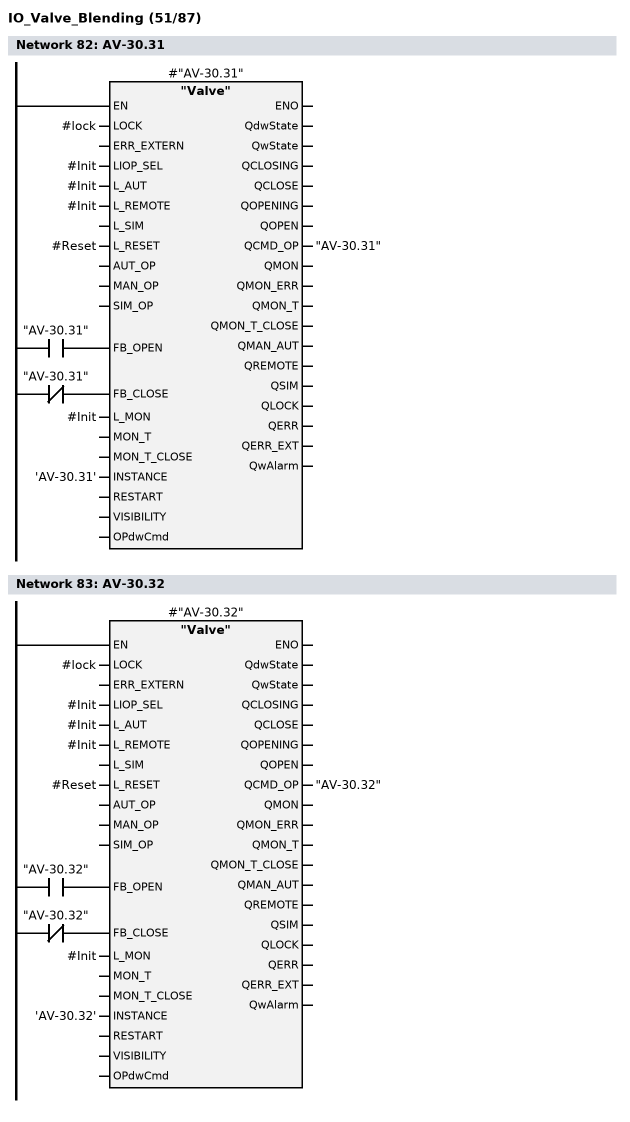
   RUNG wire#powerrail
      #"AV-30.31"(FB_OPEN := wire#w1, FB_CLOSE := wire#w2, LOCK := #lock, ERR_EXTERN :=, LIOP_SEL := #Init, L_AUT := #Init, L_REMOTE := #Init, L_SIM :=, L_RESET := #Reset, AUT_OP :=, MAN_OP :=, SIM_OP :=, L_MON := #Init, MON_T :=, MON_T_CLOSE :=, INSTANCE := 'AV-30.31', RESTART :=, VISIBILITY :=, OPdwCmd :=, QdwState =>, QwState =>, QCLOSING =>, QCLOSE =>, QOPENING =>, QOPEN =>, QCMD_OP => "AV-30.31", QMON =>, QMON_ERR =>, QMON_T =>, QMON_T_CLOSE =>, QMAN_AUT =>, QREMOTE =>, QSIM =>, QLOCK =>, QERR =>, QERR_EXT =>, QwAlarm =>)
   END_RUNG
   RUNG wire#powerrail
      Contact( "AV-30.31" )
   END_RUNG wire#w1
   RUNG wire#powerrail
      I_Contact( "AV-30.31" )
   END_RUNG wire#w2
   // the same network as SCL:
   #"AV-30.31"(LOCK := #lock,   // "Valve"
               LIOP_SEL := #Init,
               L_AUT := #Init,
               L_REMOTE := #Init,
               L_RESET := #Reset,
               FB_OPEN := "AV-30.31",
               FB_CLOSE := NOT "AV-30.31",
               L_MON := #Init,
               INSTANCE := 'AV-30.31',
               QCMD_OP => "AV-30.31");
END_REGION

REGION Network 83: AV-30.32
   RUNG wire#powerrail
      #"AV-30.32"(FB_OPEN := wire#w1, FB_CLOSE := wire#w2, LOCK := #lock, ERR_EXTERN :=, LIOP_SEL := #Init, L_AUT := #Init, L_REMOTE := #Init, L_SIM :=, L_RESET := #Reset, AUT_OP :=, MAN_OP :=, SIM_OP :=, L_MON := #Init, MON_T :=, MON_T_CLOSE :=, INSTANCE := 'AV-30.32', RESTART :=, VISIBILITY :=, OPdwCmd :=, QdwState =>, QwState =>, QCLOSING =>, QCLOSE =>, QOPENING =>, QOPEN =>, QCMD_OP => "AV-30.32", QMON =>, QMON_ERR =>, QMON_T =>, QMON_T_CLOSE =>, QMAN_AUT =>, QREMOTE =>, QSIM =>, QLOCK =>, QERR =>, QERR_EXT =>, QwAlarm =>)
   END_RUNG
   RUNG wire#powerrail
      Contact( "AV-30.32" )
   END_RUNG wire#w1
   RUNG wire#powerrail
      I_Contact( "AV-30.32" )
   END_RUNG wire#w2
   // the same network as SCL:
   #"AV-30.32"(LOCK := #lock,   // "Valve"
               LIOP_SEL := #Init,
               L_AUT := #Init,
               L_REMOTE := #Init,
               L_RESET := #Reset,
               FB_OPEN := "AV-30.32",
               FB_CLOSE := NOT "AV-30.32",
               L_MON := #Init,
               INSTANCE := 'AV-30.32',
               QCMD_OP => "AV-30.32");
END_REGION

REGION Network 84: AV-30.33
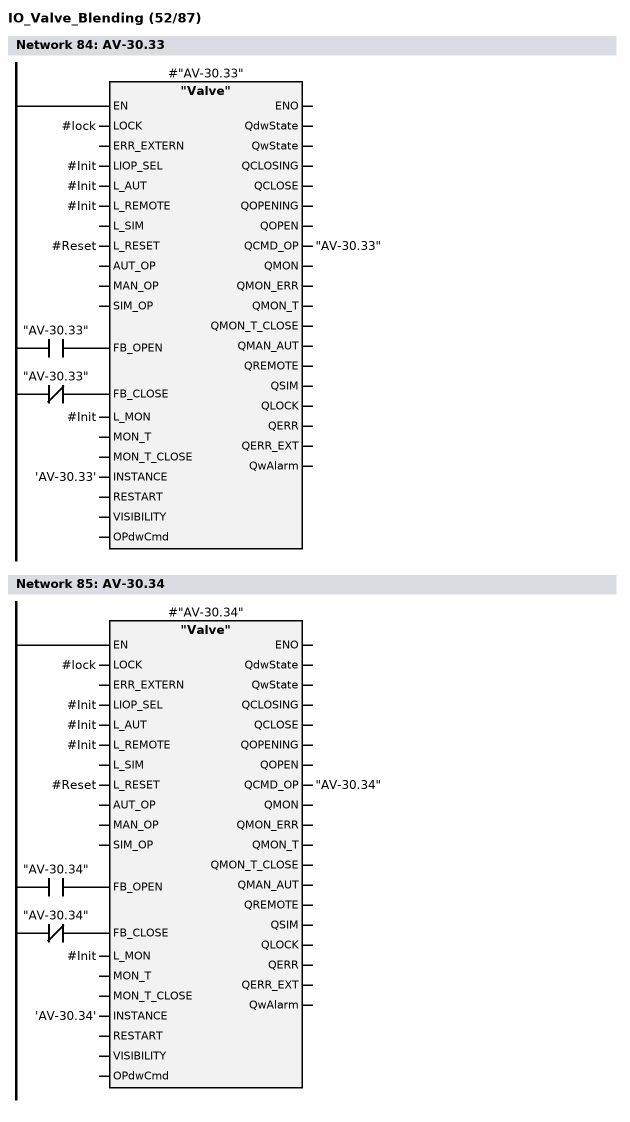
   RUNG wire#powerrail
      #"AV-30.33"(FB_OPEN := wire#w1, FB_CLOSE := wire#w2, LOCK := #lock, ERR_EXTERN :=, LIOP_SEL := #Init, L_AUT := #Init, L_REMOTE := #Init, L_SIM :=, L_RESET := #Reset, AUT_OP :=, MAN_OP :=, SIM_OP :=, L_MON := #Init, MON_T :=, MON_T_CLOSE :=, INSTANCE := 'AV-30.33', RESTART :=, VISIBILITY :=, OPdwCmd :=, QdwState =>, QwState =>, QCLOSING =>, QCLOSE =>, QOPENING =>, QOPEN =>, QCMD_OP => "AV-30.33", QMON =>, QMON_ERR =>, QMON_T =>, QMON_T_CLOSE =>, QMAN_AUT =>, QREMOTE =>, QSIM =>, QLOCK =>, QERR =>, QERR_EXT =>, QwAlarm =>)
   END_RUNG
   RUNG wire#powerrail
      Contact( "AV-30.33" )
   END_RUNG wire#w1
   RUNG wire#powerrail
      I_Contact( "AV-30.33" )
   END_RUNG wire#w2
   // the same network as SCL:
   #"AV-30.33"(LOCK := #lock,   // "Valve"
               LIOP_SEL := #Init,
               L_AUT := #Init,
               L_REMOTE := #Init,
               L_RESET := #Reset,
               FB_OPEN := "AV-30.33",
               FB_CLOSE := NOT "AV-30.33",
               L_MON := #Init,
               INSTANCE := 'AV-30.33',
               QCMD_OP => "AV-30.33");
END_REGION

REGION Network 85: AV-30.34
   RUNG wire#powerrail
      #"AV-30.34"(FB_OPEN := wire#w1, FB_CLOSE := wire#w2, LOCK := #lock, ERR_EXTERN :=, LIOP_SEL := #Init, L_AUT := #Init, L_REMOTE := #Init, L_SIM :=, L_RESET := #Reset, AUT_OP :=, MAN_OP :=, SIM_OP :=, L_MON := #Init, MON_T :=, MON_T_CLOSE :=, INSTANCE := 'AV-30.34', RESTART :=, VISIBILITY :=, OPdwCmd :=, QdwState =>, QwState =>, QCLOSING =>, QCLOSE =>, QOPENING =>, QOPEN =>, QCMD_OP => "AV-30.34", QMON =>, QMON_ERR =>, QMON_T =>, QMON_T_CLOSE =>, QMAN_AUT =>, QREMOTE =>, QSIM =>, QLOCK =>, QERR =>, QERR_EXT =>, QwAlarm =>)
   END_RUNG
   RUNG wire#powerrail
      Contact( "AV-30.34" )
   END_RUNG wire#w1
   RUNG wire#powerrail
      I_Contact( "AV-30.34" )
   END_RUNG wire#w2
   // the same network as SCL:
   #"AV-30.34"(LOCK := #lock,   // "Valve"
               LIOP_SEL := #Init,
               L_AUT := #Init,
               L_REMOTE := #Init,
               L_RESET := #Reset,
               FB_OPEN := "AV-30.34",
               FB_CLOSE := NOT "AV-30.34",
               L_MON := #Init,
               INSTANCE := 'AV-30.34',
               QCMD_OP => "AV-30.34");
END_REGION

REGION Network 86: AV-30.35
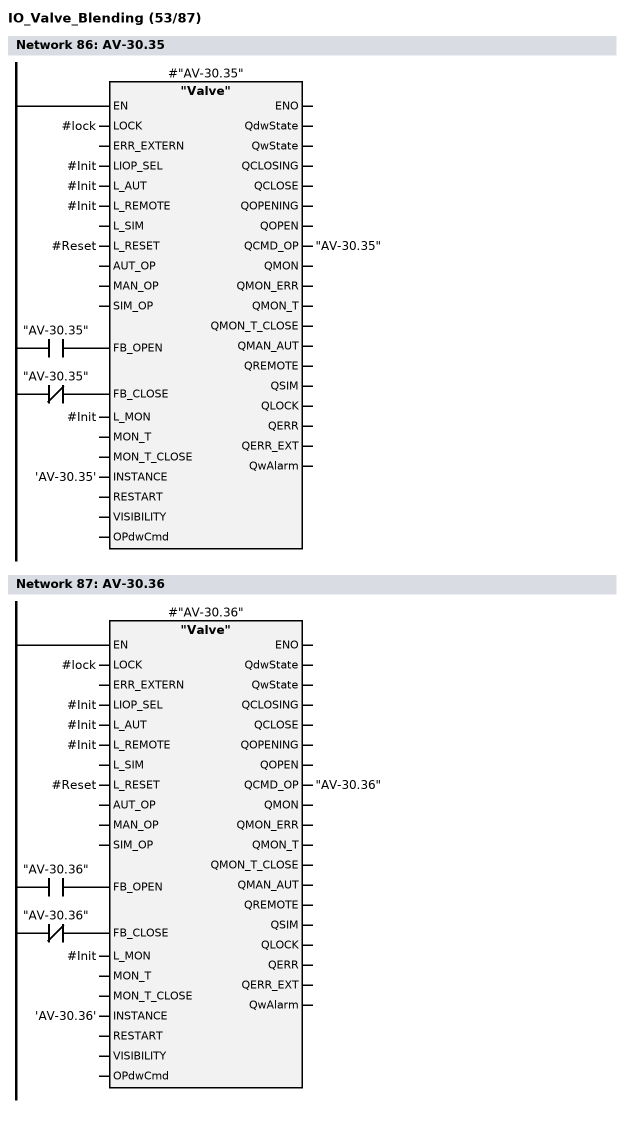
   RUNG wire#powerrail
      #"AV-30.35"(FB_OPEN := wire#w1, FB_CLOSE := wire#w2, LOCK := #lock, ERR_EXTERN :=, LIOP_SEL := #Init, L_AUT := #Init, L_REMOTE := #Init, L_SIM :=, L_RESET := #Reset, AUT_OP :=, MAN_OP :=, SIM_OP :=, L_MON := #Init, MON_T :=, MON_T_CLOSE :=, INSTANCE := 'AV-30.35', RESTART :=, VISIBILITY :=, OPdwCmd :=, QdwState =>, QwState =>, QCLOSING =>, QCLOSE =>, QOPENING =>, QOPEN =>, QCMD_OP => "AV-30.35", QMON =>, QMON_ERR =>, QMON_T =>, QMON_T_CLOSE =>, QMAN_AUT =>, QREMOTE =>, QSIM =>, QLOCK =>, QERR =>, QERR_EXT =>, QwAlarm =>)
   END_RUNG
   RUNG wire#powerrail
      Contact( "AV-30.35" )
   END_RUNG wire#w1
   RUNG wire#powerrail
      I_Contact( "AV-30.35" )
   END_RUNG wire#w2
   // the same network as SCL:
   #"AV-30.35"(LOCK := #lock,   // "Valve"
               LIOP_SEL := #Init,
               L_AUT := #Init,
               L_REMOTE := #Init,
               L_RESET := #Reset,
               FB_OPEN := "AV-30.35",
               FB_CLOSE := NOT "AV-30.35",
               L_MON := #Init,
               INSTANCE := 'AV-30.35',
               QCMD_OP => "AV-30.35");
END_REGION

REGION Network 87: AV-30.36
   RUNG wire#powerrail
      #"AV-30.36"(FB_OPEN := wire#w1, FB_CLOSE := wire#w2, LOCK := #lock, ERR_EXTERN :=, LIOP_SEL := #Init, L_AUT := #Init, L_REMOTE := #Init, L_SIM :=, L_RESET := #Reset, AUT_OP :=, MAN_OP :=, SIM_OP :=, L_MON := #Init, MON_T :=, MON_T_CLOSE :=, INSTANCE := 'AV-30.36', RESTART :=, VISIBILITY :=, OPdwCmd :=, QdwState =>, QwState =>, QCLOSING =>, QCLOSE =>, QOPENING =>, QOPEN =>, QCMD_OP => "AV-30.36", QMON =>, QMON_ERR =>, QMON_T =>, QMON_T_CLOSE =>, QMAN_AUT =>, QREMOTE =>, QSIM =>, QLOCK =>, QERR =>, QERR_EXT =>, QwAlarm =>)
   END_RUNG
   RUNG wire#powerrail
      Contact( "AV-30.36" )
   END_RUNG wire#w1
   RUNG wire#powerrail
      I_Contact( "AV-30.36" )
   END_RUNG wire#w2
   // the same network as SCL:
   #"AV-30.36"(LOCK := #lock,   // "Valve"
               LIOP_SEL := #Init,
               L_AUT := #Init,
               L_REMOTE := #Init,
               L_RESET := #Reset,
               FB_OPEN := "AV-30.36",
               FB_CLOSE := NOT "AV-30.36",
               L_MON := #Init,
               INSTANCE := 'AV-30.36',
               QCMD_OP => "AV-30.36");
END_REGION

REGION Network 88: AV-30.37
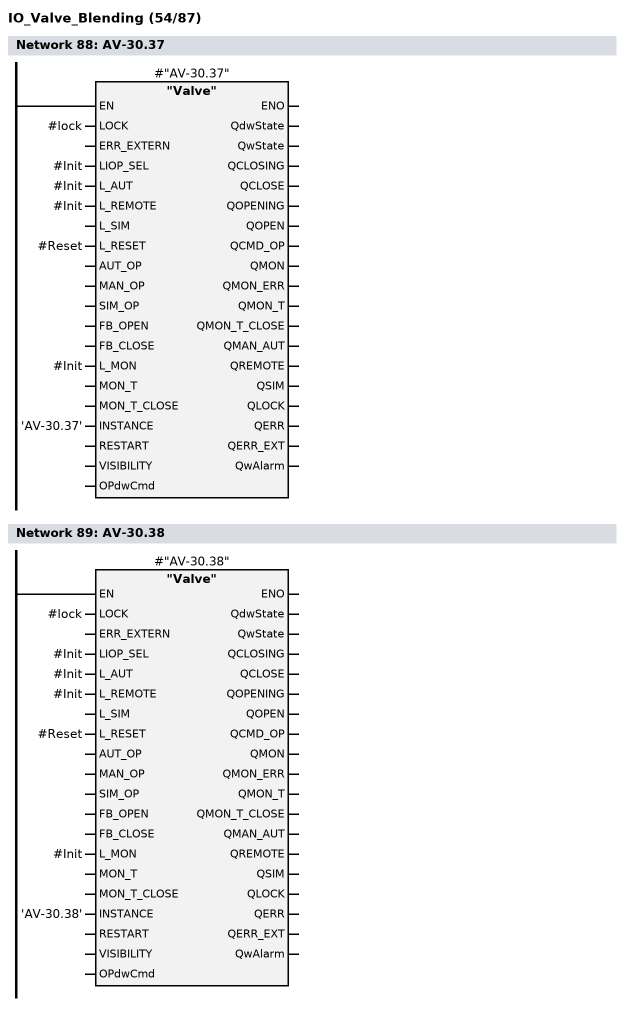
   RUNG wire#powerrail
      #"AV-30.37"(LOCK := #lock, ERR_EXTERN :=, LIOP_SEL := #Init, L_AUT := #Init, L_REMOTE := #Init, L_SIM :=, L_RESET := #Reset, AUT_OP :=, MAN_OP :=, SIM_OP :=, FB_OPEN :=, FB_CLOSE :=, L_MON := #Init, MON_T :=, MON_T_CLOSE :=, INSTANCE := 'AV-30.37', RESTART :=, VISIBILITY :=, OPdwCmd :=, QdwState =>, QwState =>, QCLOSING =>, QCLOSE =>, QOPENING =>, QOPEN =>, QCMD_OP =>, QMON =>, QMON_ERR =>, QMON_T =>, QMON_T_CLOSE =>, QMAN_AUT =>, QREMOTE =>, QSIM =>, QLOCK =>, QERR =>, QERR_EXT =>, QwAlarm =>)
   END_RUNG
   // the same network as SCL:
   #"AV-30.37"(LOCK := #lock,   // "Valve"
               LIOP_SEL := #Init,
               L_AUT := #Init,
               L_REMOTE := #Init,
               L_RESET := #Reset,
               L_MON := #Init,
               INSTANCE := 'AV-30.37');
END_REGION

REGION Network 89: AV-30.38
   RUNG wire#powerrail
      #"AV-30.38"(LOCK := #lock, ERR_EXTERN :=, LIOP_SEL := #Init, L_AUT := #Init, L_REMOTE := #Init, L_SIM :=, L_RESET := #Reset, AUT_OP :=, MAN_OP :=, SIM_OP :=, FB_OPEN :=, FB_CLOSE :=, L_MON := #Init, MON_T :=, MON_T_CLOSE :=, INSTANCE := 'AV-30.38', RESTART :=, VISIBILITY :=, OPdwCmd :=, QdwState =>, QwState =>, QCLOSING =>, QCLOSE =>, QOPENING =>, QOPEN =>, QCMD_OP =>, QMON =>, QMON_ERR =>, QMON_T =>, QMON_T_CLOSE =>, QMAN_AUT =>, QREMOTE =>, QSIM =>, QLOCK =>, QERR =>, QERR_EXT =>, QwAlarm =>)
   END_RUNG
   // the same network as SCL:
   #"AV-30.38"(LOCK := #lock,   // "Valve"
               LIOP_SEL := #Init,
               L_AUT := #Init,
               L_REMOTE := #Init,
               L_RESET := #Reset,
               L_MON := #Init,
               INSTANCE := 'AV-30.38');
END_REGION

REGION Network 90: AV-30.39
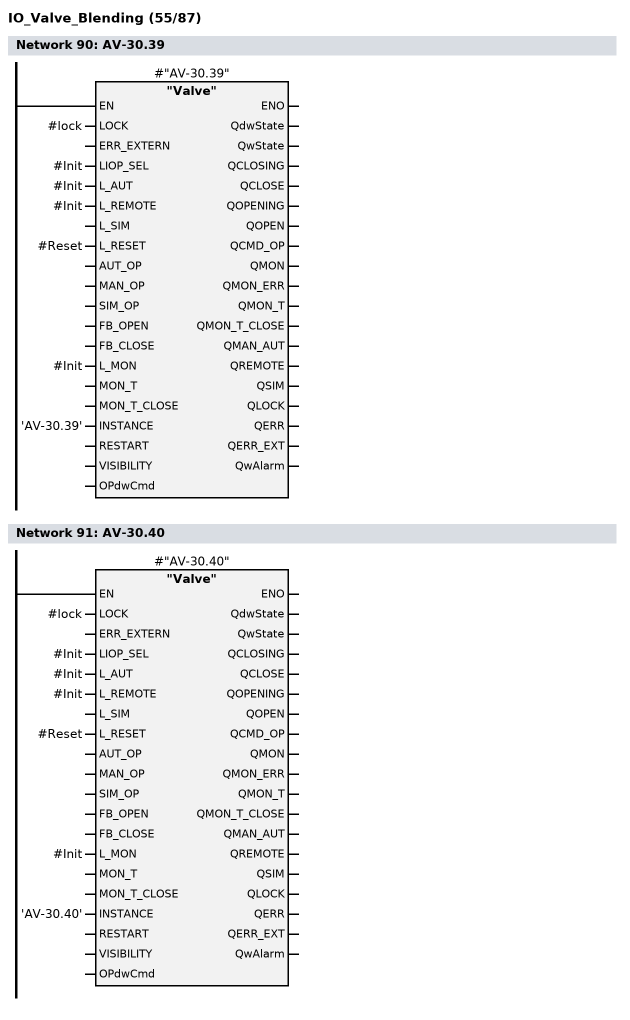
   RUNG wire#powerrail
      #"AV-30.39"(LOCK := #lock, ERR_EXTERN :=, LIOP_SEL := #Init, L_AUT := #Init, L_REMOTE := #Init, L_SIM :=, L_RESET := #Reset, AUT_OP :=, MAN_OP :=, SIM_OP :=, FB_OPEN :=, FB_CLOSE :=, L_MON := #Init, MON_T :=, MON_T_CLOSE :=, INSTANCE := 'AV-30.39', RESTART :=, VISIBILITY :=, OPdwCmd :=, QdwState =>, QwState =>, QCLOSING =>, QCLOSE =>, QOPENING =>, QOPEN =>, QCMD_OP =>, QMON =>, QMON_ERR =>, QMON_T =>, QMON_T_CLOSE =>, QMAN_AUT =>, QREMOTE =>, QSIM =>, QLOCK =>, QERR =>, QERR_EXT =>, QwAlarm =>)
   END_RUNG
   // the same network as SCL:
   #"AV-30.39"(LOCK := #lock,   // "Valve"
               LIOP_SEL := #Init,
               L_AUT := #Init,
               L_REMOTE := #Init,
               L_RESET := #Reset,
               L_MON := #Init,
               INSTANCE := 'AV-30.39');
END_REGION

REGION Network 91: AV-30.40
   RUNG wire#powerrail
      #"AV-30.40"(LOCK := #lock, ERR_EXTERN :=, LIOP_SEL := #Init, L_AUT := #Init, L_REMOTE := #Init, L_SIM :=, L_RESET := #Reset, AUT_OP :=, MAN_OP :=, SIM_OP :=, FB_OPEN :=, FB_CLOSE :=, L_MON := #Init, MON_T :=, MON_T_CLOSE :=, INSTANCE := 'AV-30.40', RESTART :=, VISIBILITY :=, OPdwCmd :=, QdwState =>, QwState =>, QCLOSING =>, QCLOSE =>, QOPENING =>, QOPEN =>, QCMD_OP =>, QMON =>, QMON_ERR =>, QMON_T =>, QMON_T_CLOSE =>, QMAN_AUT =>, QREMOTE =>, QSIM =>, QLOCK =>, QERR =>, QERR_EXT =>, QwAlarm =>)
   END_RUNG
   // the same network as SCL:
   #"AV-30.40"(LOCK := #lock,   // "Valve"
               LIOP_SEL := #Init,
               L_AUT := #Init,
               L_REMOTE := #Init,
               L_RESET := #Reset,
               L_MON := #Init,
               INSTANCE := 'AV-30.40');
END_REGION

REGION Network 92: AV-30.41
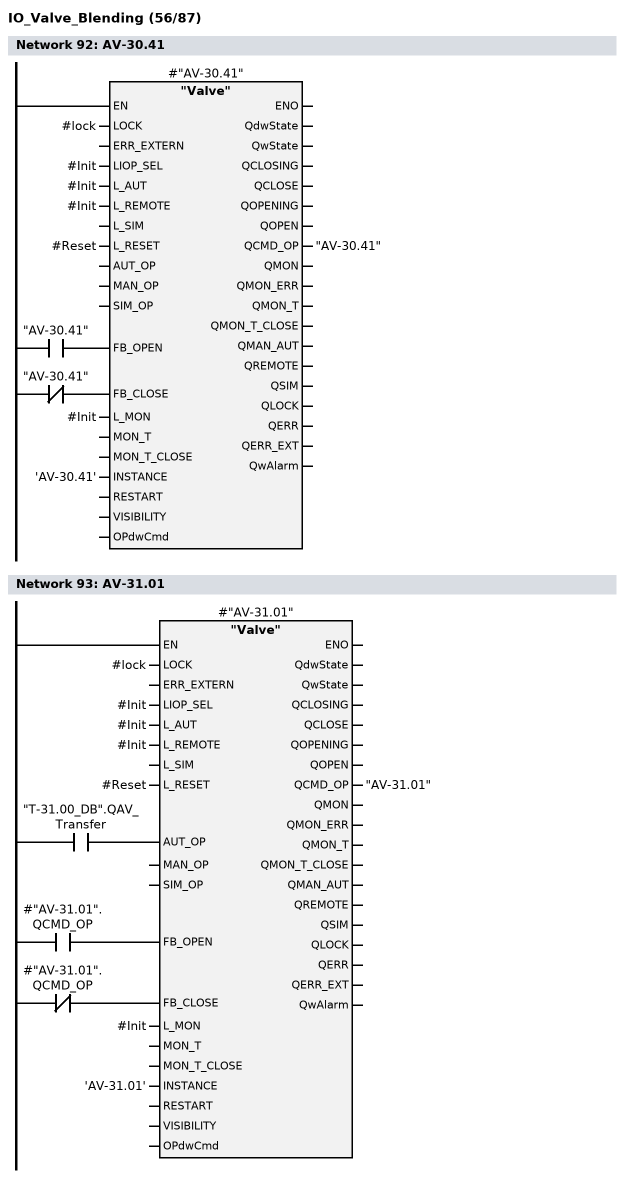
   RUNG wire#powerrail
      #"AV-30.41"(FB_OPEN := wire#w1, FB_CLOSE := wire#w2, LOCK := #lock, ERR_EXTERN :=, LIOP_SEL := #Init, L_AUT := #Init, L_REMOTE := #Init, L_SIM :=, L_RESET := #Reset, AUT_OP :=, MAN_OP :=, SIM_OP :=, L_MON := #Init, MON_T :=, MON_T_CLOSE :=, INSTANCE := 'AV-30.41', RESTART :=, VISIBILITY :=, OPdwCmd :=, QdwState =>, QwState =>, QCLOSING =>, QCLOSE =>, QOPENING =>, QOPEN =>, QCMD_OP => "AV-30.41", QMON =>, QMON_ERR =>, QMON_T =>, QMON_T_CLOSE =>, QMAN_AUT =>, QREMOTE =>, QSIM =>, QLOCK =>, QERR =>, QERR_EXT =>, QwAlarm =>)
   END_RUNG
   RUNG wire#powerrail
      Contact( "AV-30.41" )
   END_RUNG wire#w1
   RUNG wire#powerrail
      I_Contact( "AV-30.41" )
   END_RUNG wire#w2
   // the same network as SCL:
   #"AV-30.41"(LOCK := #lock,   // "Valve"
               LIOP_SEL := #Init,
               L_AUT := #Init,
               L_REMOTE := #Init,
               L_RESET := #Reset,
               FB_OPEN := "AV-30.41",
               FB_CLOSE := NOT "AV-30.41",
               L_MON := #Init,
               INSTANCE := 'AV-30.41',
               QCMD_OP => "AV-30.41");
END_REGION

REGION Network 93: AV-31.01
   RUNG wire#powerrail
      #"AV-31.01"(AUT_OP := wire#w1, FB_OPEN := wire#w2, FB_CLOSE := wire#w3, LOCK := #lock, ERR_EXTERN :=, LIOP_SEL := #Init, L_AUT := #Init, L_REMOTE := #Init, L_SIM :=, L_RESET := #Reset, MAN_OP :=, SIM_OP :=, L_MON := #Init, MON_T :=, MON_T_CLOSE :=, INSTANCE := 'AV-31.01', RESTART :=, VISIBILITY :=, OPdwCmd :=, QdwState =>, QwState =>, QCLOSING =>, QCLOSE =>, QOPENING =>, QOPEN =>, QCMD_OP => "AV-31.01", QMON =>, QMON_ERR =>, QMON_T =>, QMON_T_CLOSE =>, QMAN_AUT =>, QREMOTE =>, QSIM =>, QLOCK =>, QERR =>, QERR_EXT =>, QwAlarm =>)
   END_RUNG
   RUNG wire#powerrail
      Contact( "T-31.00_DB".QAV_Transfer )
   END_RUNG wire#w1
   RUNG wire#powerrail
      Contact( #"AV-31.01".QCMD_OP )
   END_RUNG wire#w2
   RUNG wire#powerrail
      I_Contact( #"AV-31.01".QCMD_OP )
   END_RUNG wire#w3
   // the same network as SCL:
   #"AV-31.01"(LOCK := #lock,   // "Valve"
               LIOP_SEL := #Init,
               L_AUT := #Init,
               L_REMOTE := #Init,
               L_RESET := #Reset,
               AUT_OP := "T-31.00_DB".QAV_Transfer,
               FB_OPEN := #"AV-31.01".QCMD_OP,
               FB_CLOSE := NOT #"AV-31.01".QCMD_OP,
               L_MON := #Init,
               INSTANCE := 'AV-31.01',
               QCMD_OP => "AV-31.01");
END_REGION

REGION Network 94: AV-31.02
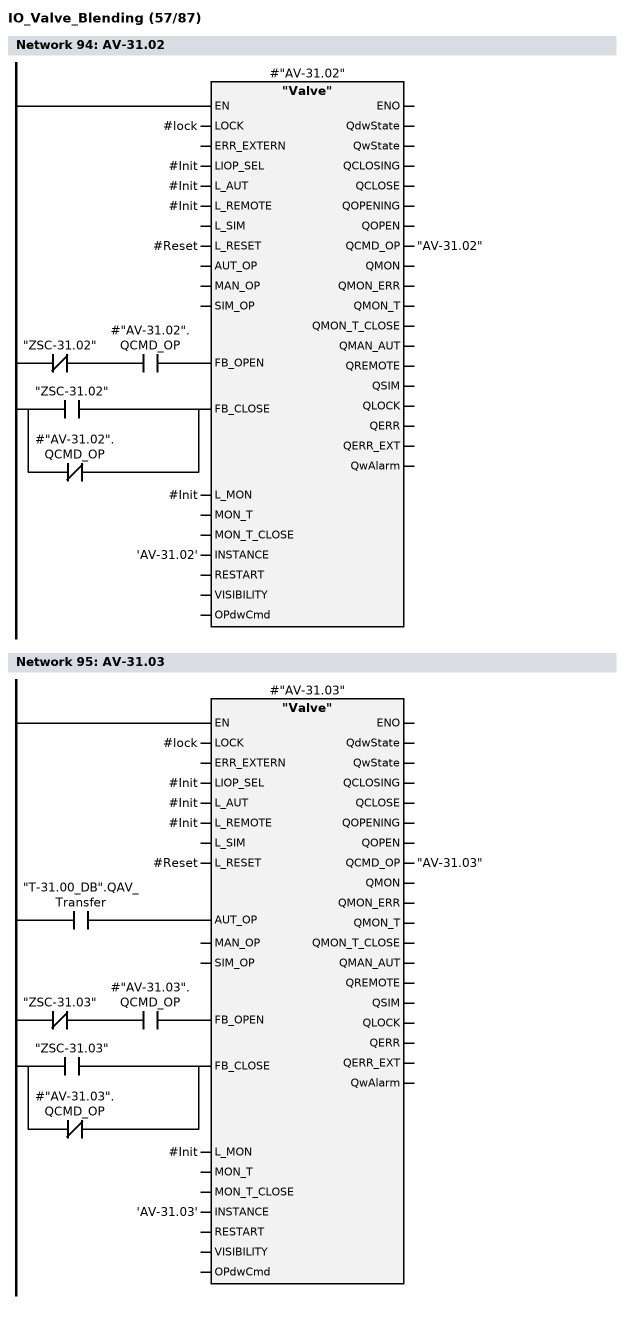
   RUNG wire#powerrail
      #"AV-31.02"(FB_OPEN := wire#w1, FB_CLOSE := wire#w2, LOCK := #lock, ERR_EXTERN :=, LIOP_SEL := #Init, L_AUT := #Init, L_REMOTE := #Init, L_SIM :=, L_RESET := #Reset, AUT_OP :=, MAN_OP :=, SIM_OP :=, L_MON := #Init, MON_T :=, MON_T_CLOSE :=, INSTANCE := 'AV-31.02', RESTART :=, VISIBILITY :=, OPdwCmd :=, QdwState =>, QwState =>, QCLOSING =>, QCLOSE =>, QOPENING =>, QOPEN =>, QCMD_OP => "AV-31.02", QMON =>, QMON_ERR =>, QMON_T =>, QMON_T_CLOSE =>, QMAN_AUT =>, QREMOTE =>, QSIM =>, QLOCK =>, QERR =>, QERR_EXT =>, QwAlarm =>)
   END_RUNG
   RUNG wire#powerrail
      I_Contact( "ZSC-31.02" )
      Contact( #"AV-31.02".QCMD_OP )
   END_RUNG wire#w1
   RUNG wire#powerrail
      Contact( "ZSC-31.02" )
   END_RUNG wire#w2
   RUNG wire#powerrail
      I_Contact( #"AV-31.02".QCMD_OP )
   END_RUNG wire#w2
   // the same network as SCL:
   #"AV-31.02"(LOCK := #lock,   // "Valve"
               LIOP_SEL := #Init,
               L_AUT := #Init,
               L_REMOTE := #Init,
               L_RESET := #Reset,
               FB_OPEN := NOT "ZSC-31.02" AND #"AV-31.02".QCMD_OP,
               FB_CLOSE := "ZSC-31.02" OR NOT #"AV-31.02".QCMD_OP,
               L_MON := #Init,
               INSTANCE := 'AV-31.02',
               QCMD_OP => "AV-31.02");
END_REGION

REGION Network 95: AV-31.03
   RUNG wire#powerrail
      #"AV-31.03"(AUT_OP := wire#w1, FB_OPEN := wire#w2, FB_CLOSE := wire#w3, LOCK := #lock, ERR_EXTERN :=, LIOP_SEL := #Init, L_AUT := #Init, L_REMOTE := #Init, L_SIM :=, L_RESET := #Reset, MAN_OP :=, SIM_OP :=, L_MON := #Init, MON_T :=, MON_T_CLOSE :=, INSTANCE := 'AV-31.03', RESTART :=, VISIBILITY :=, OPdwCmd :=, QdwState =>, QwState =>, QCLOSING =>, QCLOSE =>, QOPENING =>, QOPEN =>, QCMD_OP => "AV-31.03", QMON =>, QMON_ERR =>, QMON_T =>, QMON_T_CLOSE =>, QMAN_AUT =>, QREMOTE =>, QSIM =>, QLOCK =>, QERR =>, QERR_EXT =>, QwAlarm =>)
   END_RUNG
   RUNG wire#powerrail
      Contact( "T-31.00_DB".QAV_Transfer )
   END_RUNG wire#w1
   RUNG wire#powerrail
      I_Contact( "ZSC-31.03" )
      Contact( #"AV-31.03".QCMD_OP )
   END_RUNG wire#w2
   RUNG wire#powerrail
      Contact( "ZSC-31.03" )
   END_RUNG wire#w3
   RUNG wire#powerrail
      I_Contact( #"AV-31.03".QCMD_OP )
   END_RUNG wire#w3
   // the same network as SCL:
   #"AV-31.03"(LOCK := #lock,   // "Valve"
               LIOP_SEL := #Init,
               L_AUT := #Init,
               L_REMOTE := #Init,
               L_RESET := #Reset,
               AUT_OP := "T-31.00_DB".QAV_Transfer,
               FB_OPEN := NOT "ZSC-31.03" AND #"AV-31.03".QCMD_OP,
               FB_CLOSE := "ZSC-31.03" OR NOT #"AV-31.03".QCMD_OP,
               L_MON := #Init,
               INSTANCE := 'AV-31.03',
               QCMD_OP => "AV-31.03");
END_REGION

REGION Network 96: AV-31.04
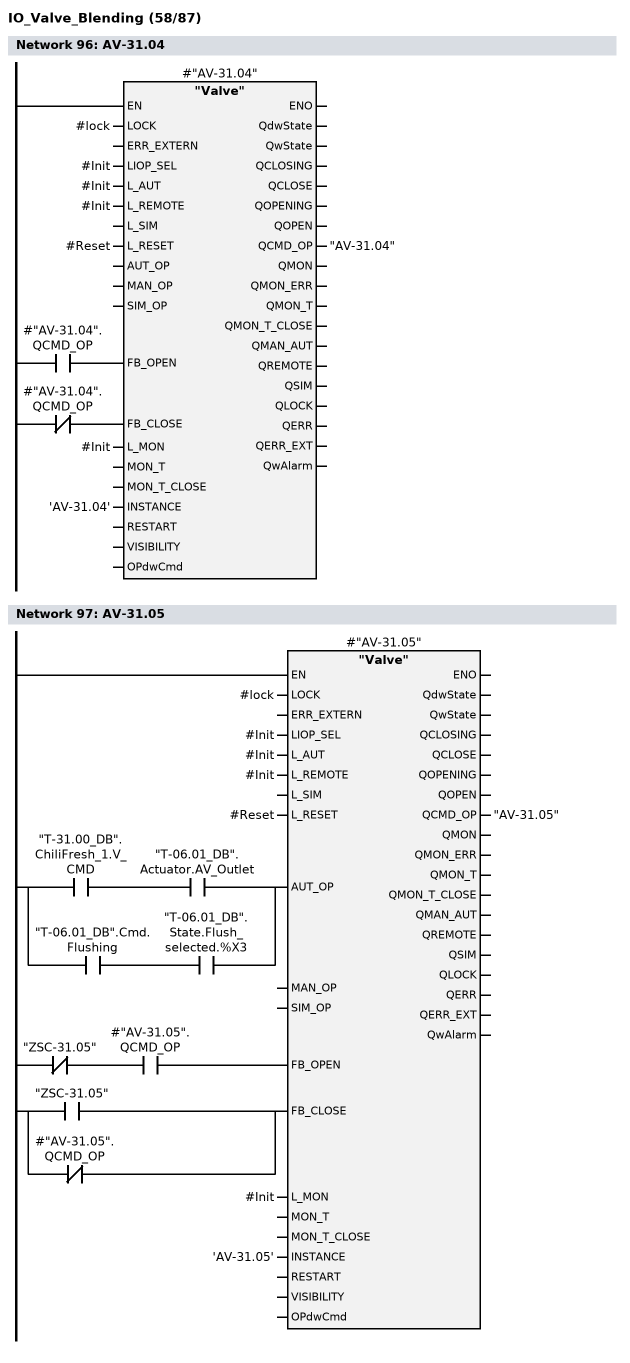
   RUNG wire#powerrail
      #"AV-31.04"(FB_OPEN := wire#w1, FB_CLOSE := wire#w2, LOCK := #lock, ERR_EXTERN :=, LIOP_SEL := #Init, L_AUT := #Init, L_REMOTE := #Init, L_SIM :=, L_RESET := #Reset, AUT_OP :=, MAN_OP :=, SIM_OP :=, L_MON := #Init, MON_T :=, MON_T_CLOSE :=, INSTANCE := 'AV-31.04', RESTART :=, VISIBILITY :=, OPdwCmd :=, QdwState =>, QwState =>, QCLOSING =>, QCLOSE =>, QOPENING =>, QOPEN =>, QCMD_OP => "AV-31.04", QMON =>, QMON_ERR =>, QMON_T =>, QMON_T_CLOSE =>, QMAN_AUT =>, QREMOTE =>, QSIM =>, QLOCK =>, QERR =>, QERR_EXT =>, QwAlarm =>)
   END_RUNG
   RUNG wire#powerrail
      Contact( #"AV-31.04".QCMD_OP )
   END_RUNG wire#w1
   RUNG wire#powerrail
      I_Contact( #"AV-31.04".QCMD_OP )
   END_RUNG wire#w2
   // the same network as SCL:
   #"AV-31.04"(LOCK := #lock,   // "Valve"
               LIOP_SEL := #Init,
               L_AUT := #Init,
               L_REMOTE := #Init,
               L_RESET := #Reset,
               FB_OPEN := #"AV-31.04".QCMD_OP,
               FB_CLOSE := NOT #"AV-31.04".QCMD_OP,
               L_MON := #Init,
               INSTANCE := 'AV-31.04',
               QCMD_OP => "AV-31.04");
END_REGION

REGION Network 97: AV-31.05
   RUNG wire#powerrail
      #"AV-31.05"(AUT_OP := wire#w1, FB_OPEN := wire#w2, FB_CLOSE := wire#w3, LOCK := #lock, ERR_EXTERN :=, LIOP_SEL := #Init, L_AUT := #Init, L_REMOTE := #Init, L_SIM :=, L_RESET := #Reset, MAN_OP :=, SIM_OP :=, L_MON := #Init, MON_T :=, MON_T_CLOSE :=, INSTANCE := 'AV-31.05', RESTART :=, VISIBILITY :=, OPdwCmd :=, QdwState =>, QwState =>, QCLOSING =>, QCLOSE =>, QOPENING =>, QOPEN =>, QCMD_OP => "AV-31.05", QMON =>, QMON_ERR =>, QMON_T =>, QMON_T_CLOSE =>, QMAN_AUT =>, QREMOTE =>, QSIM =>, QLOCK =>, QERR =>, QERR_EXT =>, QwAlarm =>)
   END_RUNG
   RUNG wire#powerrail
      Contact( "T-31.00_DB".ChiliFresh_1.V_CMD )
      Contact( "T-06.01_DB".Actuator.AV_Outlet )
   END_RUNG wire#w1
   RUNG wire#powerrail
      Contact( "T-06.01_DB".Cmd.Flushing )
      Contact( "T-06.01_DB".State.Flush_selected.%X3 )
   END_RUNG wire#w1
   RUNG wire#powerrail
      I_Contact( "ZSC-31.05" )
      Contact( #"AV-31.05".QCMD_OP )
   END_RUNG wire#w2
   RUNG wire#powerrail
      Contact( "ZSC-31.05" )
   END_RUNG wire#w3
   RUNG wire#powerrail
      I_Contact( #"AV-31.05".QCMD_OP )
   END_RUNG wire#w3
   // the same network as SCL:
   #"AV-31.05"(LOCK := #lock,   // "Valve"
               LIOP_SEL := #Init,
               L_AUT := #Init,
               L_REMOTE := #Init,
               L_RESET := #Reset,
               AUT_OP := ("T-31.00_DB".ChiliFresh_1.V_CMD AND "T-06.01_DB".Actuator.AV_Outlet) OR ("T-06.01_DB".Cmd.Flushing AND "T-06.01_DB".State.Flush_selected.%X3),
               FB_OPEN := NOT "ZSC-31.05" AND #"AV-31.05".QCMD_OP,
               FB_CLOSE := "ZSC-31.05" OR NOT #"AV-31.05".QCMD_OP,
               L_MON := #Init,
               INSTANCE := 'AV-31.05',
               QCMD_OP => "AV-31.05");
END_REGION

REGION Network 98: AV-31.06
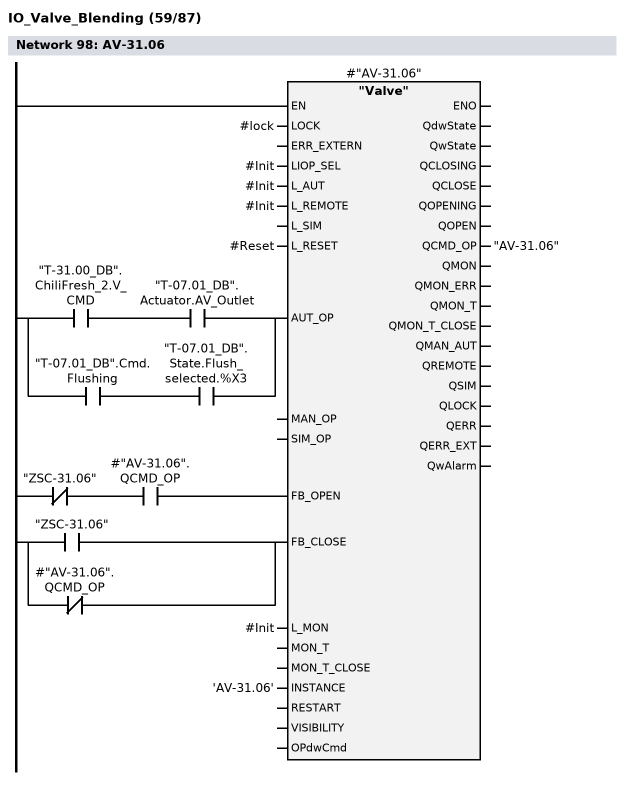
   RUNG wire#powerrail
      #"AV-31.06"(AUT_OP := wire#w1, FB_OPEN := wire#w2, FB_CLOSE := wire#w3, LOCK := #lock, ERR_EXTERN :=, LIOP_SEL := #Init, L_AUT := #Init, L_REMOTE := #Init, L_SIM :=, L_RESET := #Reset, MAN_OP :=, SIM_OP :=, L_MON := #Init, MON_T :=, MON_T_CLOSE :=, INSTANCE := 'AV-31.06', RESTART :=, VISIBILITY :=, OPdwCmd :=, QdwState =>, QwState =>, QCLOSING =>, QCLOSE =>, QOPENING =>, QOPEN =>, QCMD_OP => "AV-31.06", QMON =>, QMON_ERR =>, QMON_T =>, QMON_T_CLOSE =>, QMAN_AUT =>, QREMOTE =>, QSIM =>, QLOCK =>, QERR =>, QERR_EXT =>, QwAlarm =>)
   END_RUNG
   RUNG wire#powerrail
      Contact( "T-31.00_DB".ChiliFresh_2.V_CMD )
      Contact( "T-07.01_DB".Actuator.AV_Outlet )
   END_RUNG wire#w1
   RUNG wire#powerrail
      Contact( "T-07.01_DB".Cmd.Flushing )
      Contact( "T-07.01_DB".State.Flush_selected.%X3 )
   END_RUNG wire#w1
   RUNG wire#powerrail
      I_Contact( "ZSC-31.06" )
      Contact( #"AV-31.06".QCMD_OP )
   END_RUNG wire#w2
   RUNG wire#powerrail
      Contact( "ZSC-31.06" )
   END_RUNG wire#w3
   RUNG wire#powerrail
      I_Contact( #"AV-31.06".QCMD_OP )
   END_RUNG wire#w3
   // the same network as SCL:
   #"AV-31.06"(LOCK := #lock,   // "Valve"
               LIOP_SEL := #Init,
               L_AUT := #Init,
               L_REMOTE := #Init,
               L_RESET := #Reset,
               AUT_OP := ("T-31.00_DB".ChiliFresh_2.V_CMD AND "T-07.01_DB".Actuator.AV_Outlet) OR ("T-07.01_DB".Cmd.Flushing AND "T-07.01_DB".State.Flush_selected.%X3),
               FB_OPEN := NOT "ZSC-31.06" AND #"AV-31.06".QCMD_OP,
               FB_CLOSE := "ZSC-31.06" OR NOT #"AV-31.06".QCMD_OP,
               L_MON := #Init,
               INSTANCE := 'AV-31.06',
               QCMD_OP => "AV-31.06");
END_REGION

REGION Network 99: AV-31.07
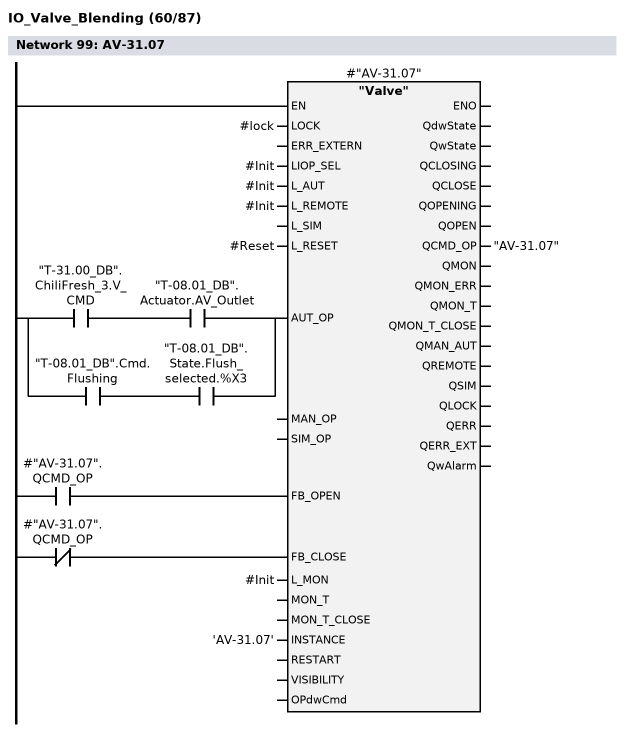
   RUNG wire#powerrail
      #"AV-31.07"(AUT_OP := wire#w1, FB_OPEN := wire#w2, FB_CLOSE := wire#w3, LOCK := #lock, ERR_EXTERN :=, LIOP_SEL := #Init, L_AUT := #Init, L_REMOTE := #Init, L_SIM :=, L_RESET := #Reset, MAN_OP :=, SIM_OP :=, L_MON := #Init, MON_T :=, MON_T_CLOSE :=, INSTANCE := 'AV-31.07', RESTART :=, VISIBILITY :=, OPdwCmd :=, QdwState =>, QwState =>, QCLOSING =>, QCLOSE =>, QOPENING =>, QOPEN =>, QCMD_OP => "AV-31.07", QMON =>, QMON_ERR =>, QMON_T =>, QMON_T_CLOSE =>, QMAN_AUT =>, QREMOTE =>, QSIM =>, QLOCK =>, QERR =>, QERR_EXT =>, QwAlarm =>)
   END_RUNG
   RUNG wire#powerrail
      Contact( "T-31.00_DB".ChiliFresh_3.V_CMD )
      Contact( "T-08.01_DB".Actuator.AV_Outlet )
   END_RUNG wire#w1
   RUNG wire#powerrail
      Contact( "T-08.01_DB".Cmd.Flushing )
      Contact( "T-08.01_DB".State.Flush_selected.%X3 )
   END_RUNG wire#w1
   RUNG wire#powerrail
      Contact( #"AV-31.07".QCMD_OP )
   END_RUNG wire#w2
   RUNG wire#powerrail
      I_Contact( #"AV-31.07".QCMD_OP )
   END_RUNG wire#w3
   // the same network as SCL:
   #"AV-31.07"(LOCK := #lock,   // "Valve"
               LIOP_SEL := #Init,
               L_AUT := #Init,
               L_REMOTE := #Init,
               L_RESET := #Reset,
               AUT_OP := ("T-31.00_DB".ChiliFresh_3.V_CMD AND "T-08.01_DB".Actuator.AV_Outlet) OR ("T-08.01_DB".Cmd.Flushing AND "T-08.01_DB".State.Flush_selected.%X3),
               FB_OPEN := #"AV-31.07".QCMD_OP,
               FB_CLOSE := NOT #"AV-31.07".QCMD_OP,
               L_MON := #Init,
               INSTANCE := 'AV-31.07',
               QCMD_OP => "AV-31.07");
END_REGION

REGION Network 100: AV-31.08
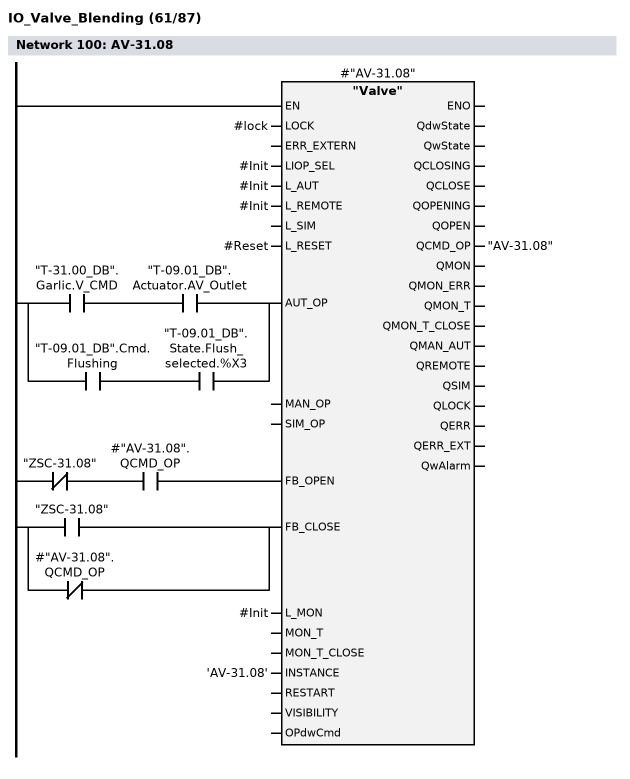
   RUNG wire#powerrail
      #"AV-31.08"(AUT_OP := wire#w1, FB_OPEN := wire#w2, FB_CLOSE := wire#w3, LOCK := #lock, ERR_EXTERN :=, LIOP_SEL := #Init, L_AUT := #Init, L_REMOTE := #Init, L_SIM :=, L_RESET := #Reset, MAN_OP :=, SIM_OP :=, L_MON := #Init, MON_T :=, MON_T_CLOSE :=, INSTANCE := 'AV-31.08', RESTART :=, VISIBILITY :=, OPdwCmd :=, QdwState =>, QwState =>, QCLOSING =>, QCLOSE =>, QOPENING =>, QOPEN =>, QCMD_OP => "AV-31.08", QMON =>, QMON_ERR =>, QMON_T =>, QMON_T_CLOSE =>, QMAN_AUT =>, QREMOTE =>, QSIM =>, QLOCK =>, QERR =>, QERR_EXT =>, QwAlarm =>)
   END_RUNG
   RUNG wire#powerrail
      Contact( "T-31.00_DB".Garlic.V_CMD )
      Contact( "T-09.01_DB".Actuator.AV_Outlet )
   END_RUNG wire#w1
   RUNG wire#powerrail
      Contact( "T-09.01_DB".Cmd.Flushing )
      Contact( "T-09.01_DB".State.Flush_selected.%X3 )
   END_RUNG wire#w1
   RUNG wire#powerrail
      I_Contact( "ZSC-31.08" )
      Contact( #"AV-31.08".QCMD_OP )
   END_RUNG wire#w2
   RUNG wire#powerrail
      Contact( "ZSC-31.08" )
   END_RUNG wire#w3
   RUNG wire#powerrail
      I_Contact( #"AV-31.08".QCMD_OP )
   END_RUNG wire#w3
   // the same network as SCL:
   #"AV-31.08"(LOCK := #lock,   // "Valve"
               LIOP_SEL := #Init,
               L_AUT := #Init,
               L_REMOTE := #Init,
               L_RESET := #Reset,
               AUT_OP := ("T-31.00_DB".Garlic.V_CMD AND "T-09.01_DB".Actuator.AV_Outlet) OR ("T-09.01_DB".Cmd.Flushing AND "T-09.01_DB".State.Flush_selected.%X3),
               FB_OPEN := NOT "ZSC-31.08" AND #"AV-31.08".QCMD_OP,
               FB_CLOSE := "ZSC-31.08" OR NOT #"AV-31.08".QCMD_OP,
               L_MON := #Init,
               INSTANCE := 'AV-31.08',
               QCMD_OP => "AV-31.08");
END_REGION

REGION Network 101: AV-31.09
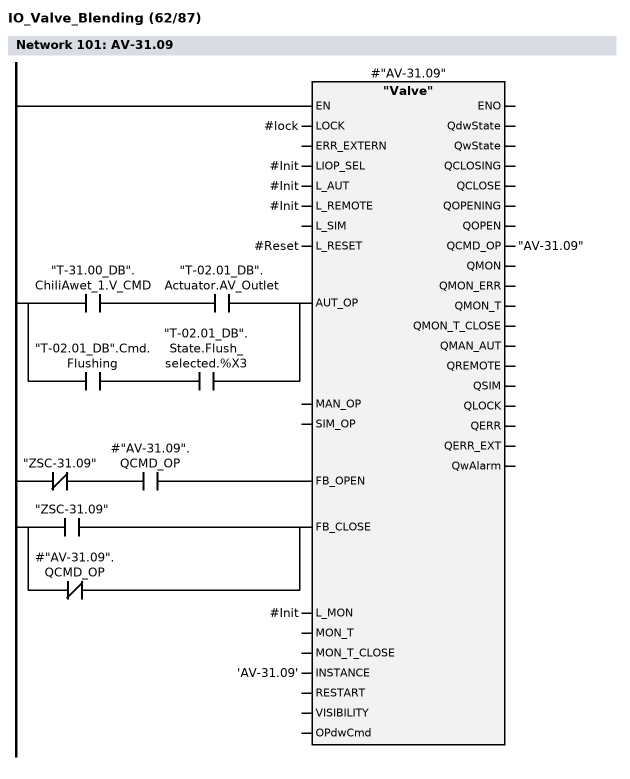
   RUNG wire#powerrail
      #"AV-31.09"(AUT_OP := wire#w1, FB_OPEN := wire#w2, FB_CLOSE := wire#w3, LOCK := #lock, ERR_EXTERN :=, LIOP_SEL := #Init, L_AUT := #Init, L_REMOTE := #Init, L_SIM :=, L_RESET := #Reset, MAN_OP :=, SIM_OP :=, L_MON := #Init, MON_T :=, MON_T_CLOSE :=, INSTANCE := 'AV-31.09', RESTART :=, VISIBILITY :=, OPdwCmd :=, QdwState =>, QwState =>, QCLOSING =>, QCLOSE =>, QOPENING =>, QOPEN =>, QCMD_OP => "AV-31.09", QMON =>, QMON_ERR =>, QMON_T =>, QMON_T_CLOSE =>, QMAN_AUT =>, QREMOTE =>, QSIM =>, QLOCK =>, QERR =>, QERR_EXT =>, QwAlarm =>)
   END_RUNG
   RUNG wire#powerrail
      Contact( "T-31.00_DB".ChiliAwet_1.V_CMD )
      Contact( "T-02.01_DB".Actuator.AV_Outlet )
   END_RUNG wire#w1
   RUNG wire#powerrail
      Contact( "T-02.01_DB".Cmd.Flushing )
      Contact( "T-02.01_DB".State.Flush_selected.%X3 )
   END_RUNG wire#w1
   RUNG wire#powerrail
      I_Contact( "ZSC-31.09" )
      Contact( #"AV-31.09".QCMD_OP )
   END_RUNG wire#w2
   RUNG wire#powerrail
      Contact( "ZSC-31.09" )
   END_RUNG wire#w3
   RUNG wire#powerrail
      I_Contact( #"AV-31.09".QCMD_OP )
   END_RUNG wire#w3
   // the same network as SCL:
   #"AV-31.09"(LOCK := #lock,   // "Valve"
               LIOP_SEL := #Init,
               L_AUT := #Init,
               L_REMOTE := #Init,
               L_RESET := #Reset,
               AUT_OP := ("T-31.00_DB".ChiliAwet_1.V_CMD AND "T-02.01_DB".Actuator.AV_Outlet) OR ("T-02.01_DB".Cmd.Flushing AND "T-02.01_DB".State.Flush_selected.%X3),
               FB_OPEN := NOT "ZSC-31.09" AND #"AV-31.09".QCMD_OP,
               FB_CLOSE := "ZSC-31.09" OR NOT #"AV-31.09".QCMD_OP,
               L_MON := #Init,
               INSTANCE := 'AV-31.09',
               QCMD_OP => "AV-31.09");
END_REGION

REGION Network 102: AV-31.10
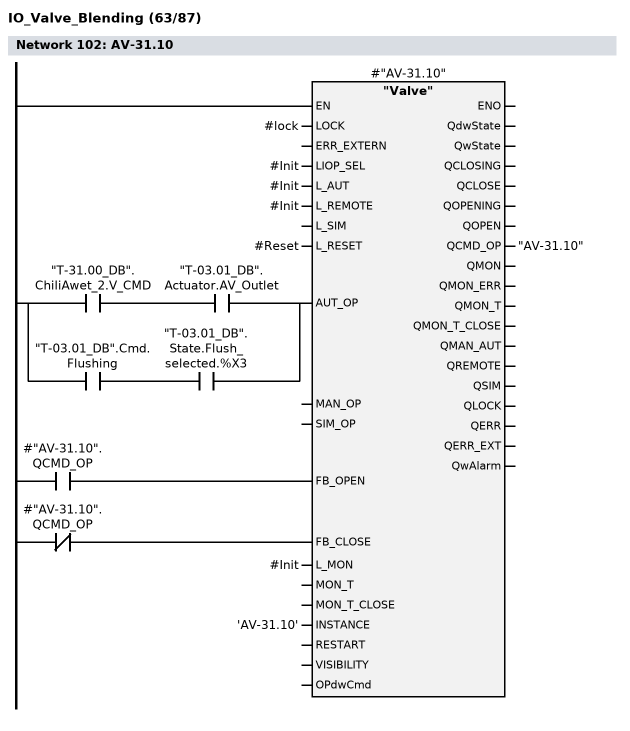
   RUNG wire#powerrail
      #"AV-31.10"(AUT_OP := wire#w1, FB_OPEN := wire#w2, FB_CLOSE := wire#w3, LOCK := #lock, ERR_EXTERN :=, LIOP_SEL := #Init, L_AUT := #Init, L_REMOTE := #Init, L_SIM :=, L_RESET := #Reset, MAN_OP :=, SIM_OP :=, L_MON := #Init, MON_T :=, MON_T_CLOSE :=, INSTANCE := 'AV-31.10', RESTART :=, VISIBILITY :=, OPdwCmd :=, QdwState =>, QwState =>, QCLOSING =>, QCLOSE =>, QOPENING =>, QOPEN =>, QCMD_OP => "AV-31.10", QMON =>, QMON_ERR =>, QMON_T =>, QMON_T_CLOSE =>, QMAN_AUT =>, QREMOTE =>, QSIM =>, QLOCK =>, QERR =>, QERR_EXT =>, QwAlarm =>)
   END_RUNG
   RUNG wire#powerrail
      Contact( "T-31.00_DB".ChiliAwet_2.V_CMD )
      Contact( "T-03.01_DB".Actuator.AV_Outlet )
   END_RUNG wire#w1
   RUNG wire#powerrail
      Contact( "T-03.01_DB".Cmd.Flushing )
      Contact( "T-03.01_DB".State.Flush_selected.%X3 )
   END_RUNG wire#w1
   RUNG wire#powerrail
      Contact( #"AV-31.10".QCMD_OP )
   END_RUNG wire#w2
   RUNG wire#powerrail
      I_Contact( #"AV-31.10".QCMD_OP )
   END_RUNG wire#w3
   // the same network as SCL:
   #"AV-31.10"(LOCK := #lock,   // "Valve"
               LIOP_SEL := #Init,
               L_AUT := #Init,
               L_REMOTE := #Init,
               L_RESET := #Reset,
               AUT_OP := ("T-31.00_DB".ChiliAwet_2.V_CMD AND "T-03.01_DB".Actuator.AV_Outlet) OR ("T-03.01_DB".Cmd.Flushing AND "T-03.01_DB".State.Flush_selected.%X3),
               FB_OPEN := #"AV-31.10".QCMD_OP,
               FB_CLOSE := NOT #"AV-31.10".QCMD_OP,
               L_MON := #Init,
               INSTANCE := 'AV-31.10',
               QCMD_OP => "AV-31.10");
END_REGION

REGION Network 103: AV-31.11
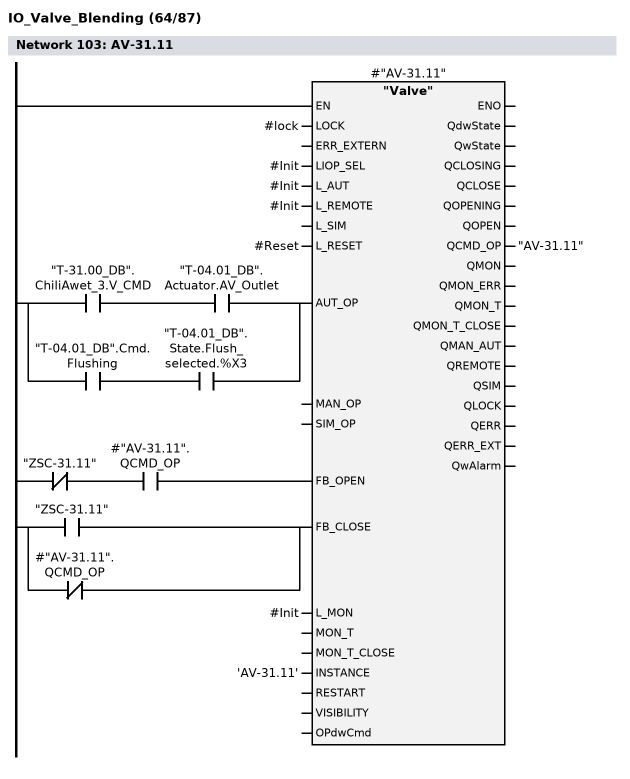
   RUNG wire#powerrail
      #"AV-31.11"(AUT_OP := wire#w1, FB_OPEN := wire#w2, FB_CLOSE := wire#w3, LOCK := #lock, ERR_EXTERN :=, LIOP_SEL := #Init, L_AUT := #Init, L_REMOTE := #Init, L_SIM :=, L_RESET := #Reset, MAN_OP :=, SIM_OP :=, L_MON := #Init, MON_T :=, MON_T_CLOSE :=, INSTANCE := 'AV-31.11', RESTART :=, VISIBILITY :=, OPdwCmd :=, QdwState =>, QwState =>, QCLOSING =>, QCLOSE =>, QOPENING =>, QOPEN =>, QCMD_OP => "AV-31.11", QMON =>, QMON_ERR =>, QMON_T =>, QMON_T_CLOSE =>, QMAN_AUT =>, QREMOTE =>, QSIM =>, QLOCK =>, QERR =>, QERR_EXT =>, QwAlarm =>)
   END_RUNG
   RUNG wire#powerrail
      Contact( "T-31.00_DB".ChiliAwet_3.V_CMD )
      Contact( "T-04.01_DB".Actuator.AV_Outlet )
   END_RUNG wire#w1
   RUNG wire#powerrail
      Contact( "T-04.01_DB".Cmd.Flushing )
      Contact( "T-04.01_DB".State.Flush_selected.%X3 )
   END_RUNG wire#w1
   RUNG wire#powerrail
      I_Contact( "ZSC-31.11" )
      Contact( #"AV-31.11".QCMD_OP )
   END_RUNG wire#w2
   RUNG wire#powerrail
      Contact( "ZSC-31.11" )
   END_RUNG wire#w3
   RUNG wire#powerrail
      I_Contact( #"AV-31.11".QCMD_OP )
   END_RUNG wire#w3
   // the same network as SCL:
   #"AV-31.11"(LOCK := #lock,   // "Valve"
               LIOP_SEL := #Init,
               L_AUT := #Init,
               L_REMOTE := #Init,
               L_RESET := #Reset,
               AUT_OP := ("T-31.00_DB".ChiliAwet_3.V_CMD AND "T-04.01_DB".Actuator.AV_Outlet) OR ("T-04.01_DB".Cmd.Flushing AND "T-04.01_DB".State.Flush_selected.%X3),
               FB_OPEN := NOT "ZSC-31.11" AND #"AV-31.11".QCMD_OP,
               FB_CLOSE := "ZSC-31.11" OR NOT #"AV-31.11".QCMD_OP,
               L_MON := #Init,
               INSTANCE := 'AV-31.11',
               QCMD_OP => "AV-31.11");
END_REGION

REGION Network 104: AV-31.12
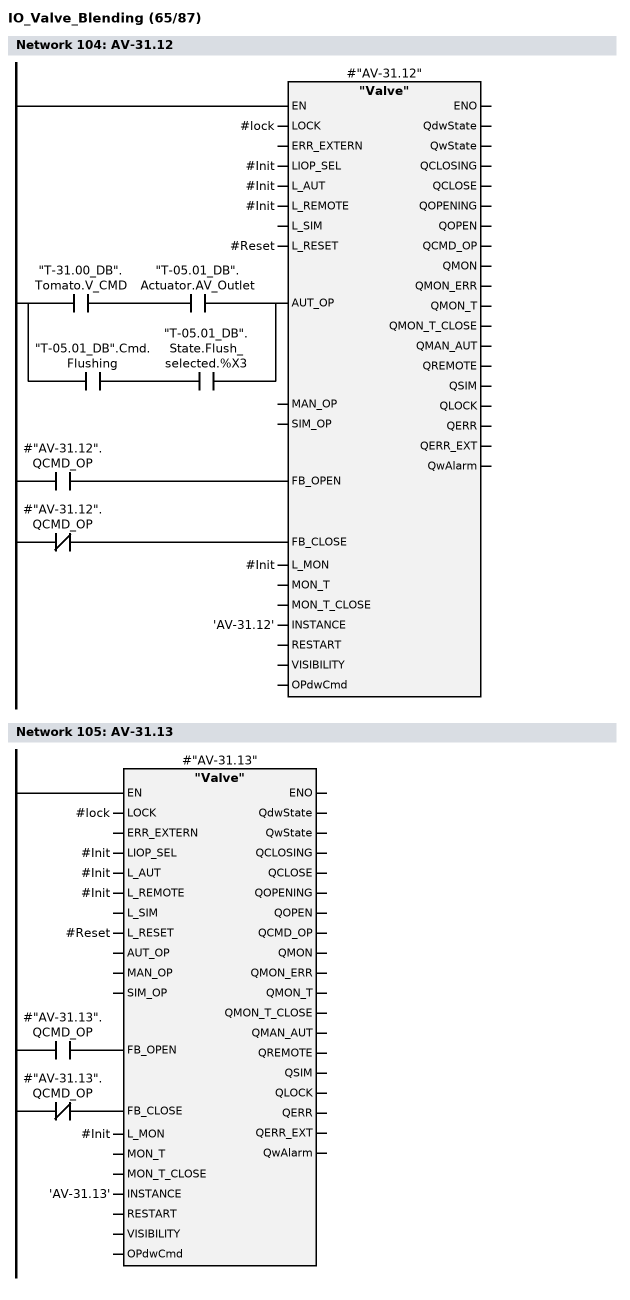
   RUNG wire#powerrail
      #"AV-31.12"(AUT_OP := wire#w1, FB_OPEN := wire#w2, FB_CLOSE := wire#w3, LOCK := #lock, ERR_EXTERN :=, LIOP_SEL := #Init, L_AUT := #Init, L_REMOTE := #Init, L_SIM :=, L_RESET := #Reset, MAN_OP :=, SIM_OP :=, L_MON := #Init, MON_T :=, MON_T_CLOSE :=, INSTANCE := 'AV-31.12', RESTART :=, VISIBILITY :=, OPdwCmd :=, QdwState =>, QwState =>, QCLOSING =>, QCLOSE =>, QOPENING =>, QOPEN =>, QCMD_OP =>, QMON =>, QMON_ERR =>, QMON_T =>, QMON_T_CLOSE =>, QMAN_AUT =>, QREMOTE =>, QSIM =>, QLOCK =>, QERR =>, QERR_EXT =>, QwAlarm =>)
   END_RUNG
   RUNG wire#powerrail
      Contact( "T-31.00_DB".Tomato.V_CMD )
      Contact( "T-05.01_DB".Actuator.AV_Outlet )
   END_RUNG wire#w1
   RUNG wire#powerrail
      Contact( "T-05.01_DB".Cmd.Flushing )
      Contact( "T-05.01_DB".State.Flush_selected.%X3 )
   END_RUNG wire#w1
   RUNG wire#powerrail
      Contact( #"AV-31.12".QCMD_OP )
   END_RUNG wire#w2
   RUNG wire#powerrail
      I_Contact( #"AV-31.12".QCMD_OP )
   END_RUNG wire#w3
   // the same network as SCL:
   #"AV-31.12"(LOCK := #lock,   // "Valve"
               LIOP_SEL := #Init,
               L_AUT := #Init,
               L_REMOTE := #Init,
               L_RESET := #Reset,
               AUT_OP := ("T-31.00_DB".Tomato.V_CMD AND "T-05.01_DB".Actuator.AV_Outlet) OR ("T-05.01_DB".Cmd.Flushing AND "T-05.01_DB".State.Flush_selected.%X3),
               FB_OPEN := #"AV-31.12".QCMD_OP,
               FB_CLOSE := NOT #"AV-31.12".QCMD_OP,
               L_MON := #Init,
               INSTANCE := 'AV-31.12');
END_REGION

REGION Network 105: AV-31.13
   RUNG wire#powerrail
      #"AV-31.13"(FB_OPEN := wire#w1, FB_CLOSE := wire#w2, LOCK := #lock, ERR_EXTERN :=, LIOP_SEL := #Init, L_AUT := #Init, L_REMOTE := #Init, L_SIM :=, L_RESET := #Reset, AUT_OP :=, MAN_OP :=, SIM_OP :=, L_MON := #Init, MON_T :=, MON_T_CLOSE :=, INSTANCE := 'AV-31.13', RESTART :=, VISIBILITY :=, OPdwCmd :=, QdwState =>, QwState =>, QCLOSING =>, QCLOSE =>, QOPENING =>, QOPEN =>, QCMD_OP =>, QMON =>, QMON_ERR =>, QMON_T =>, QMON_T_CLOSE =>, QMAN_AUT =>, QREMOTE =>, QSIM =>, QLOCK =>, QERR =>, QERR_EXT =>, QwAlarm =>)
   END_RUNG
   RUNG wire#powerrail
      Contact( #"AV-31.13".QCMD_OP )
   END_RUNG wire#w1
   RUNG wire#powerrail
      I_Contact( #"AV-31.13".QCMD_OP )
   END_RUNG wire#w2
   // the same network as SCL:
   #"AV-31.13"(LOCK := #lock,   // "Valve"
               LIOP_SEL := #Init,
               L_AUT := #Init,
               L_REMOTE := #Init,
               L_RESET := #Reset,
               FB_OPEN := #"AV-31.13".QCMD_OP,
               FB_CLOSE := NOT #"AV-31.13".QCMD_OP,
               L_MON := #Init,
               INSTANCE := 'AV-31.13');
END_REGION

REGION Network 106: AV-31.14
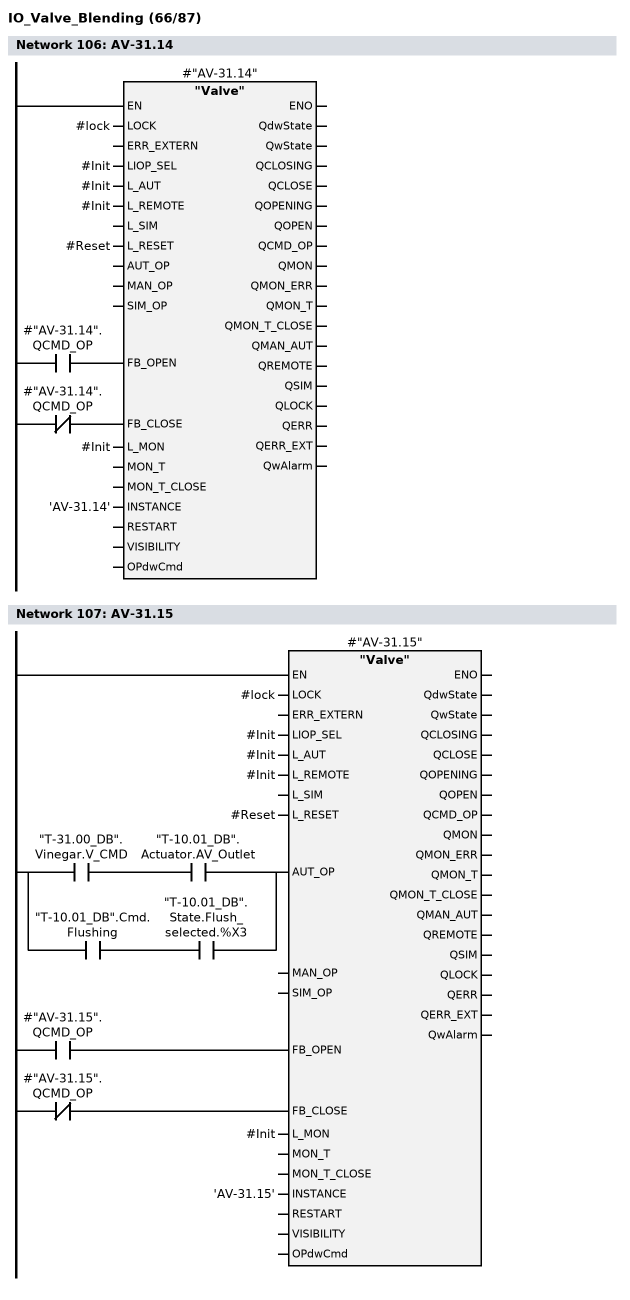
   RUNG wire#powerrail
      #"AV-31.14"(FB_OPEN := wire#w1, FB_CLOSE := wire#w2, LOCK := #lock, ERR_EXTERN :=, LIOP_SEL := #Init, L_AUT := #Init, L_REMOTE := #Init, L_SIM :=, L_RESET := #Reset, AUT_OP :=, MAN_OP :=, SIM_OP :=, L_MON := #Init, MON_T :=, MON_T_CLOSE :=, INSTANCE := 'AV-31.14', RESTART :=, VISIBILITY :=, OPdwCmd :=, QdwState =>, QwState =>, QCLOSING =>, QCLOSE =>, QOPENING =>, QOPEN =>, QCMD_OP =>, QMON =>, QMON_ERR =>, QMON_T =>, QMON_T_CLOSE =>, QMAN_AUT =>, QREMOTE =>, QSIM =>, QLOCK =>, QERR =>, QERR_EXT =>, QwAlarm =>)
   END_RUNG
   RUNG wire#powerrail
      Contact( #"AV-31.14".QCMD_OP )
   END_RUNG wire#w1
   RUNG wire#powerrail
      I_Contact( #"AV-31.14".QCMD_OP )
   END_RUNG wire#w2
   // the same network as SCL:
   #"AV-31.14"(LOCK := #lock,   // "Valve"
               LIOP_SEL := #Init,
               L_AUT := #Init,
               L_REMOTE := #Init,
               L_RESET := #Reset,
               FB_OPEN := #"AV-31.14".QCMD_OP,
               FB_CLOSE := NOT #"AV-31.14".QCMD_OP,
               L_MON := #Init,
               INSTANCE := 'AV-31.14');
END_REGION

REGION Network 107: AV-31.15
   RUNG wire#powerrail
      #"AV-31.15"(AUT_OP := wire#w1, FB_OPEN := wire#w2, FB_CLOSE := wire#w3, LOCK := #lock, ERR_EXTERN :=, LIOP_SEL := #Init, L_AUT := #Init, L_REMOTE := #Init, L_SIM :=, L_RESET := #Reset, MAN_OP :=, SIM_OP :=, L_MON := #Init, MON_T :=, MON_T_CLOSE :=, INSTANCE := 'AV-31.15', RESTART :=, VISIBILITY :=, OPdwCmd :=, QdwState =>, QwState =>, QCLOSING =>, QCLOSE =>, QOPENING =>, QOPEN =>, QCMD_OP =>, QMON =>, QMON_ERR =>, QMON_T =>, QMON_T_CLOSE =>, QMAN_AUT =>, QREMOTE =>, QSIM =>, QLOCK =>, QERR =>, QERR_EXT =>, QwAlarm =>)
   END_RUNG
   RUNG wire#powerrail
      Contact( "T-31.00_DB".Vinegar.V_CMD )
      Contact( "T-10.01_DB".Actuator.AV_Outlet )
   END_RUNG wire#w1
   RUNG wire#powerrail
      Contact( "T-10.01_DB".Cmd.Flushing )
      Contact( "T-10.01_DB".State.Flush_selected.%X3 )
   END_RUNG wire#w1
   RUNG wire#powerrail
      Contact( #"AV-31.15".QCMD_OP )
   END_RUNG wire#w2
   RUNG wire#powerrail
      I_Contact( #"AV-31.15".QCMD_OP )
   END_RUNG wire#w3
   // the same network as SCL:
   #"AV-31.15"(LOCK := #lock,   // "Valve"
               LIOP_SEL := #Init,
               L_AUT := #Init,
               L_REMOTE := #Init,
               L_RESET := #Reset,
               AUT_OP := ("T-31.00_DB".Vinegar.V_CMD AND "T-10.01_DB".Actuator.AV_Outlet) OR ("T-10.01_DB".Cmd.Flushing AND "T-10.01_DB".State.Flush_selected.%X3),
               FB_OPEN := #"AV-31.15".QCMD_OP,
               FB_CLOSE := NOT #"AV-31.15".QCMD_OP,
               L_MON := #Init,
               INSTANCE := 'AV-31.15');
END_REGION

REGION Network 108: AV-31.16
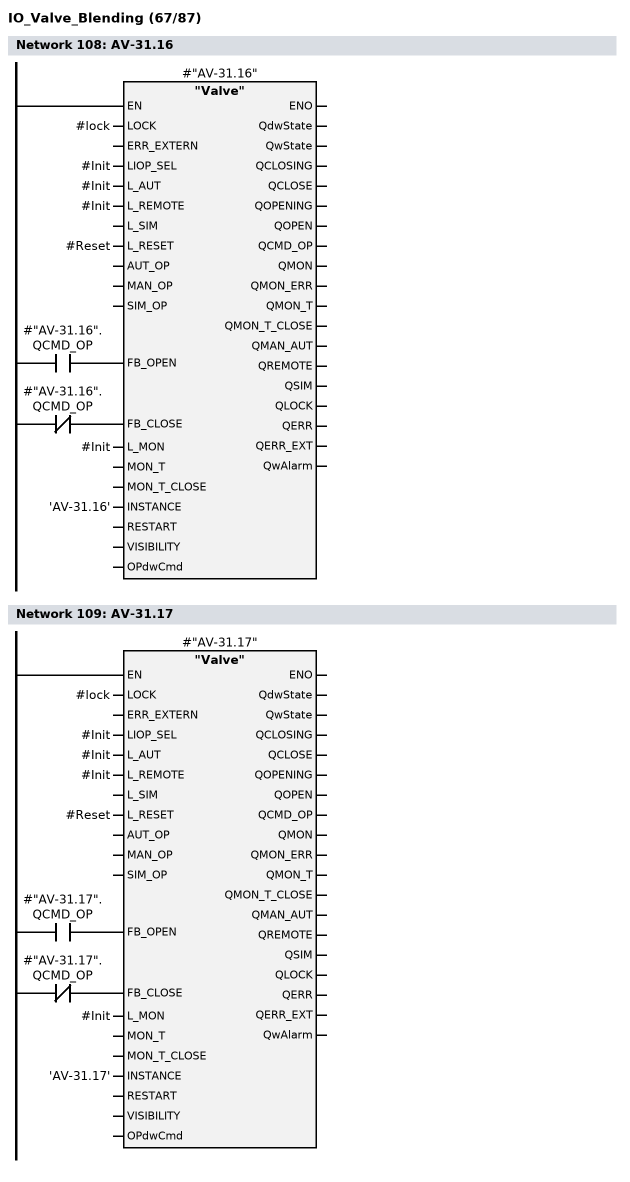
   RUNG wire#powerrail
      #"AV-31.16"(FB_OPEN := wire#w1, FB_CLOSE := wire#w2, LOCK := #lock, ERR_EXTERN :=, LIOP_SEL := #Init, L_AUT := #Init, L_REMOTE := #Init, L_SIM :=, L_RESET := #Reset, AUT_OP :=, MAN_OP :=, SIM_OP :=, L_MON := #Init, MON_T :=, MON_T_CLOSE :=, INSTANCE := 'AV-31.16', RESTART :=, VISIBILITY :=, OPdwCmd :=, QdwState =>, QwState =>, QCLOSING =>, QCLOSE =>, QOPENING =>, QOPEN =>, QCMD_OP =>, QMON =>, QMON_ERR =>, QMON_T =>, QMON_T_CLOSE =>, QMAN_AUT =>, QREMOTE =>, QSIM =>, QLOCK =>, QERR =>, QERR_EXT =>, QwAlarm =>)
   END_RUNG
   RUNG wire#powerrail
      Contact( #"AV-31.16".QCMD_OP )
   END_RUNG wire#w1
   RUNG wire#powerrail
      I_Contact( #"AV-31.16".QCMD_OP )
   END_RUNG wire#w2
   // the same network as SCL:
   #"AV-31.16"(LOCK := #lock,   // "Valve"
               LIOP_SEL := #Init,
               L_AUT := #Init,
               L_REMOTE := #Init,
               L_RESET := #Reset,
               FB_OPEN := #"AV-31.16".QCMD_OP,
               FB_CLOSE := NOT #"AV-31.16".QCMD_OP,
               L_MON := #Init,
               INSTANCE := 'AV-31.16');
END_REGION

REGION Network 109: AV-31.17
   RUNG wire#powerrail
      #"AV-31.17"(FB_OPEN := wire#w1, FB_CLOSE := wire#w2, LOCK := #lock, ERR_EXTERN :=, LIOP_SEL := #Init, L_AUT := #Init, L_REMOTE := #Init, L_SIM :=, L_RESET := #Reset, AUT_OP :=, MAN_OP :=, SIM_OP :=, L_MON := #Init, MON_T :=, MON_T_CLOSE :=, INSTANCE := 'AV-31.17', RESTART :=, VISIBILITY :=, OPdwCmd :=, QdwState =>, QwState =>, QCLOSING =>, QCLOSE =>, QOPENING =>, QOPEN =>, QCMD_OP =>, QMON =>, QMON_ERR =>, QMON_T =>, QMON_T_CLOSE =>, QMAN_AUT =>, QREMOTE =>, QSIM =>, QLOCK =>, QERR =>, QERR_EXT =>, QwAlarm =>)
   END_RUNG
   RUNG wire#powerrail
      Contact( #"AV-31.17".QCMD_OP )
   END_RUNG wire#w1
   RUNG wire#powerrail
      I_Contact( #"AV-31.17".QCMD_OP )
   END_RUNG wire#w2
   // the same network as SCL:
   #"AV-31.17"(LOCK := #lock,   // "Valve"
               LIOP_SEL := #Init,
               L_AUT := #Init,
               L_REMOTE := #Init,
               L_RESET := #Reset,
               FB_OPEN := #"AV-31.17".QCMD_OP,
               FB_CLOSE := NOT #"AV-31.17".QCMD_OP,
               L_MON := #Init,
               INSTANCE := 'AV-31.17');
END_REGION

REGION Network 110: AV-31.18
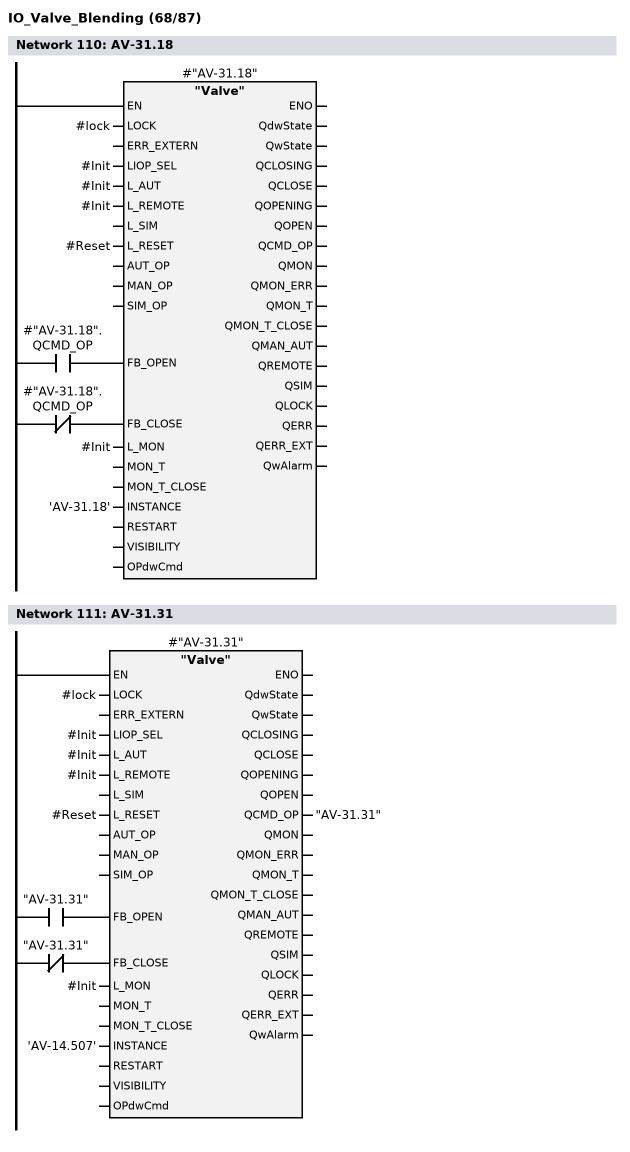
   RUNG wire#powerrail
      #"AV-31.18"(FB_OPEN := wire#w1, FB_CLOSE := wire#w2, LOCK := #lock, ERR_EXTERN :=, LIOP_SEL := #Init, L_AUT := #Init, L_REMOTE := #Init, L_SIM :=, L_RESET := #Reset, AUT_OP :=, MAN_OP :=, SIM_OP :=, L_MON := #Init, MON_T :=, MON_T_CLOSE :=, INSTANCE := 'AV-31.18', RESTART :=, VISIBILITY :=, OPdwCmd :=, QdwState =>, QwState =>, QCLOSING =>, QCLOSE =>, QOPENING =>, QOPEN =>, QCMD_OP =>, QMON =>, QMON_ERR =>, QMON_T =>, QMON_T_CLOSE =>, QMAN_AUT =>, QREMOTE =>, QSIM =>, QLOCK =>, QERR =>, QERR_EXT =>, QwAlarm =>)
   END_RUNG
   RUNG wire#powerrail
      Contact( #"AV-31.18".QCMD_OP )
   END_RUNG wire#w1
   RUNG wire#powerrail
      I_Contact( #"AV-31.18".QCMD_OP )
   END_RUNG wire#w2
   // the same network as SCL:
   #"AV-31.18"(LOCK := #lock,   // "Valve"
               LIOP_SEL := #Init,
               L_AUT := #Init,
               L_REMOTE := #Init,
               L_RESET := #Reset,
               FB_OPEN := #"AV-31.18".QCMD_OP,
               FB_CLOSE := NOT #"AV-31.18".QCMD_OP,
               L_MON := #Init,
               INSTANCE := 'AV-31.18');
END_REGION

REGION Network 111: AV-31.31
   RUNG wire#powerrail
      #"AV-31.31"(FB_OPEN := wire#w1, FB_CLOSE := wire#w2, LOCK := #lock, ERR_EXTERN :=, LIOP_SEL := #Init, L_AUT := #Init, L_REMOTE := #Init, L_SIM :=, L_RESET := #Reset, AUT_OP :=, MAN_OP :=, SIM_OP :=, L_MON := #Init, MON_T :=, MON_T_CLOSE :=, INSTANCE := 'AV-14.507', RESTART :=, VISIBILITY :=, OPdwCmd :=, QdwState =>, QwState =>, QCLOSING =>, QCLOSE =>, QOPENING =>, QOPEN =>, QCMD_OP => "AV-31.31", QMON =>, QMON_ERR =>, QMON_T =>, QMON_T_CLOSE =>, QMAN_AUT =>, QREMOTE =>, QSIM =>, QLOCK =>, QERR =>, QERR_EXT =>, QwAlarm =>)
   END_RUNG
   RUNG wire#powerrail
      Contact( "AV-31.31" )
   END_RUNG wire#w1
   RUNG wire#powerrail
      I_Contact( "AV-31.31" )
   END_RUNG wire#w2
   // the same network as SCL:
   #"AV-31.31"(LOCK := #lock,   // "Valve"
               LIOP_SEL := #Init,
               L_AUT := #Init,
               L_REMOTE := #Init,
               L_RESET := #Reset,
               FB_OPEN := "AV-31.31",
               FB_CLOSE := NOT "AV-31.31",
               L_MON := #Init,
               INSTANCE := 'AV-14.507',
               QCMD_OP => "AV-31.31");
END_REGION

REGION Network 112: AV-31.32
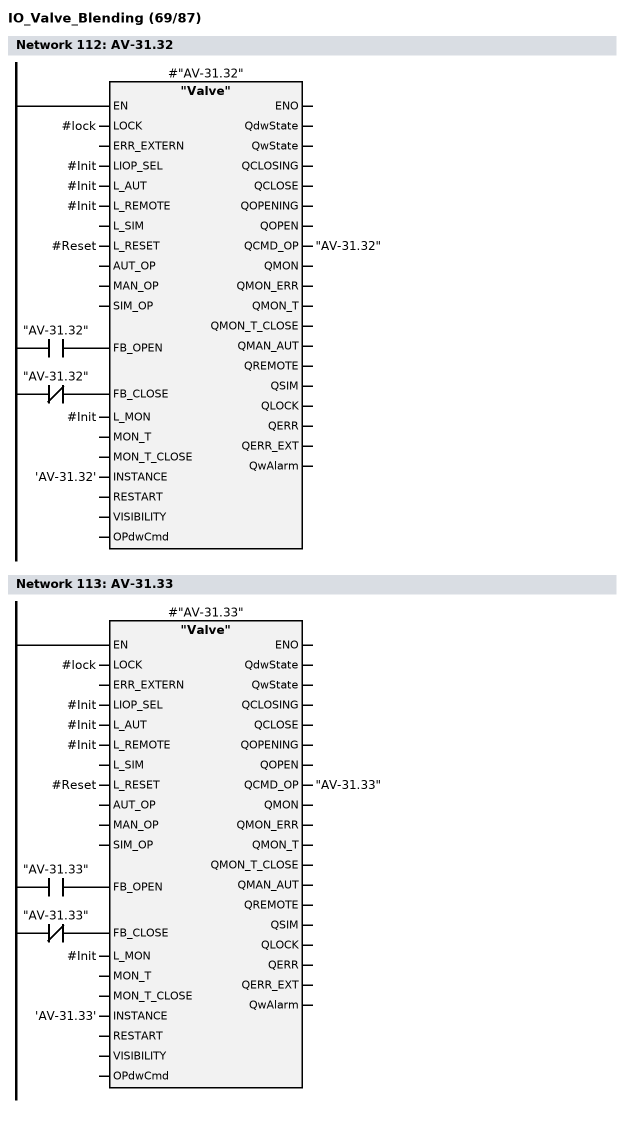
   RUNG wire#powerrail
      #"AV-31.32"(FB_OPEN := wire#w1, FB_CLOSE := wire#w2, LOCK := #lock, ERR_EXTERN :=, LIOP_SEL := #Init, L_AUT := #Init, L_REMOTE := #Init, L_SIM :=, L_RESET := #Reset, AUT_OP :=, MAN_OP :=, SIM_OP :=, L_MON := #Init, MON_T :=, MON_T_CLOSE :=, INSTANCE := 'AV-31.32', RESTART :=, VISIBILITY :=, OPdwCmd :=, QdwState =>, QwState =>, QCLOSING =>, QCLOSE =>, QOPENING =>, QOPEN =>, QCMD_OP => "AV-31.32", QMON =>, QMON_ERR =>, QMON_T =>, QMON_T_CLOSE =>, QMAN_AUT =>, QREMOTE =>, QSIM =>, QLOCK =>, QERR =>, QERR_EXT =>, QwAlarm =>)
   END_RUNG
   RUNG wire#powerrail
      Contact( "AV-31.32" )
   END_RUNG wire#w1
   RUNG wire#powerrail
      I_Contact( "AV-31.32" )
   END_RUNG wire#w2
   // the same network as SCL:
   #"AV-31.32"(LOCK := #lock,   // "Valve"
               LIOP_SEL := #Init,
               L_AUT := #Init,
               L_REMOTE := #Init,
               L_RESET := #Reset,
               FB_OPEN := "AV-31.32",
               FB_CLOSE := NOT "AV-31.32",
               L_MON := #Init,
               INSTANCE := 'AV-31.32',
               QCMD_OP => "AV-31.32");
END_REGION

REGION Network 113: AV-31.33
   RUNG wire#powerrail
      #"AV-31.33"(FB_OPEN := wire#w1, FB_CLOSE := wire#w2, LOCK := #lock, ERR_EXTERN :=, LIOP_SEL := #Init, L_AUT := #Init, L_REMOTE := #Init, L_SIM :=, L_RESET := #Reset, AUT_OP :=, MAN_OP :=, SIM_OP :=, L_MON := #Init, MON_T :=, MON_T_CLOSE :=, INSTANCE := 'AV-31.33', RESTART :=, VISIBILITY :=, OPdwCmd :=, QdwState =>, QwState =>, QCLOSING =>, QCLOSE =>, QOPENING =>, QOPEN =>, QCMD_OP => "AV-31.33", QMON =>, QMON_ERR =>, QMON_T =>, QMON_T_CLOSE =>, QMAN_AUT =>, QREMOTE =>, QSIM =>, QLOCK =>, QERR =>, QERR_EXT =>, QwAlarm =>)
   END_RUNG
   RUNG wire#powerrail
      Contact( "AV-31.33" )
   END_RUNG wire#w1
   RUNG wire#powerrail
      I_Contact( "AV-31.33" )
   END_RUNG wire#w2
   // the same network as SCL:
   #"AV-31.33"(LOCK := #lock,   // "Valve"
               LIOP_SEL := #Init,
               L_AUT := #Init,
               L_REMOTE := #Init,
               L_RESET := #Reset,
               FB_OPEN := "AV-31.33",
               FB_CLOSE := NOT "AV-31.33",
               L_MON := #Init,
               INSTANCE := 'AV-31.33',
               QCMD_OP => "AV-31.33");
END_REGION

REGION Network 114: AV-31.34
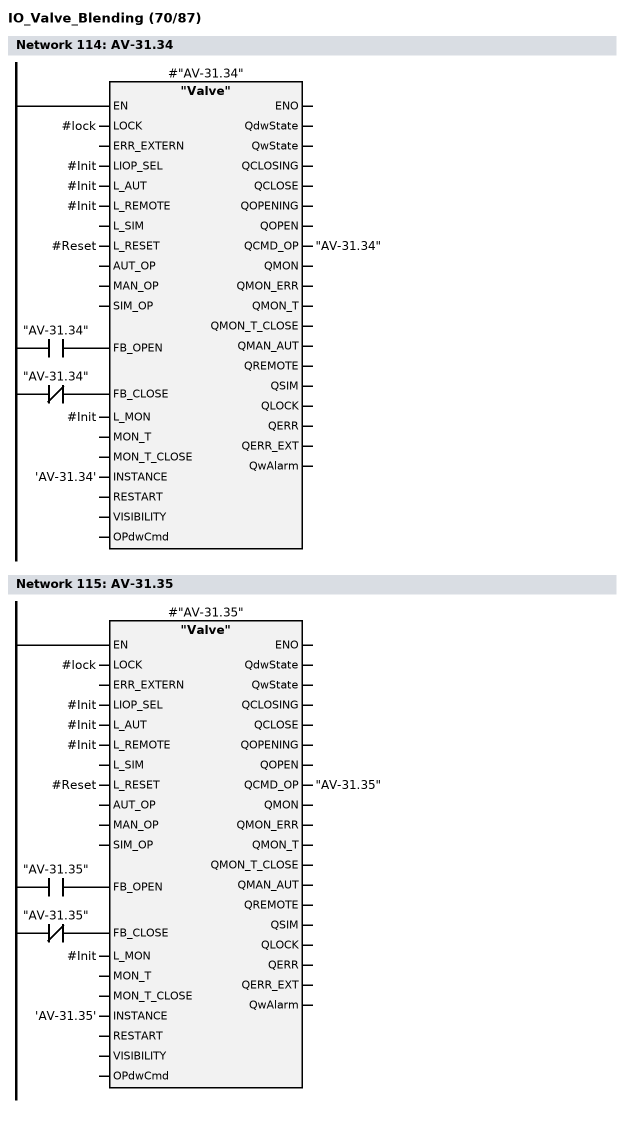
   RUNG wire#powerrail
      #"AV-31.34"(FB_OPEN := wire#w1, FB_CLOSE := wire#w2, LOCK := #lock, ERR_EXTERN :=, LIOP_SEL := #Init, L_AUT := #Init, L_REMOTE := #Init, L_SIM :=, L_RESET := #Reset, AUT_OP :=, MAN_OP :=, SIM_OP :=, L_MON := #Init, MON_T :=, MON_T_CLOSE :=, INSTANCE := 'AV-31.34', RESTART :=, VISIBILITY :=, OPdwCmd :=, QdwState =>, QwState =>, QCLOSING =>, QCLOSE =>, QOPENING =>, QOPEN =>, QCMD_OP => "AV-31.34", QMON =>, QMON_ERR =>, QMON_T =>, QMON_T_CLOSE =>, QMAN_AUT =>, QREMOTE =>, QSIM =>, QLOCK =>, QERR =>, QERR_EXT =>, QwAlarm =>)
   END_RUNG
   RUNG wire#powerrail
      Contact( "AV-31.34" )
   END_RUNG wire#w1
   RUNG wire#powerrail
      I_Contact( "AV-31.34" )
   END_RUNG wire#w2
   // the same network as SCL:
   #"AV-31.34"(LOCK := #lock,   // "Valve"
               LIOP_SEL := #Init,
               L_AUT := #Init,
               L_REMOTE := #Init,
               L_RESET := #Reset,
               FB_OPEN := "AV-31.34",
               FB_CLOSE := NOT "AV-31.34",
               L_MON := #Init,
               INSTANCE := 'AV-31.34',
               QCMD_OP => "AV-31.34");
END_REGION

REGION Network 115: AV-31.35
   RUNG wire#powerrail
      #"AV-31.35"(FB_OPEN := wire#w1, FB_CLOSE := wire#w2, LOCK := #lock, ERR_EXTERN :=, LIOP_SEL := #Init, L_AUT := #Init, L_REMOTE := #Init, L_SIM :=, L_RESET := #Reset, AUT_OP :=, MAN_OP :=, SIM_OP :=, L_MON := #Init, MON_T :=, MON_T_CLOSE :=, INSTANCE := 'AV-31.35', RESTART :=, VISIBILITY :=, OPdwCmd :=, QdwState =>, QwState =>, QCLOSING =>, QCLOSE =>, QOPENING =>, QOPEN =>, QCMD_OP => "AV-31.35", QMON =>, QMON_ERR =>, QMON_T =>, QMON_T_CLOSE =>, QMAN_AUT =>, QREMOTE =>, QSIM =>, QLOCK =>, QERR =>, QERR_EXT =>, QwAlarm =>)
   END_RUNG
   RUNG wire#powerrail
      Contact( "AV-31.35" )
   END_RUNG wire#w1
   RUNG wire#powerrail
      I_Contact( "AV-31.35" )
   END_RUNG wire#w2
   // the same network as SCL:
   #"AV-31.35"(LOCK := #lock,   // "Valve"
               LIOP_SEL := #Init,
               L_AUT := #Init,
               L_REMOTE := #Init,
               L_RESET := #Reset,
               FB_OPEN := "AV-31.35",
               FB_CLOSE := NOT "AV-31.35",
               L_MON := #Init,
               INSTANCE := 'AV-31.35',
               QCMD_OP => "AV-31.35");
END_REGION

REGION Network 116: AV-31.36
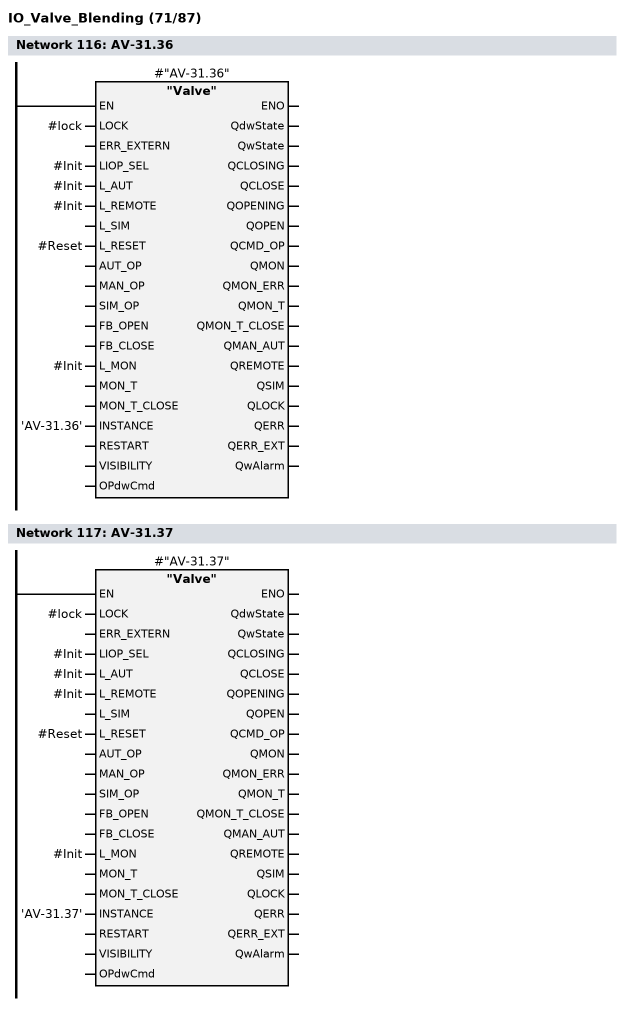
   RUNG wire#powerrail
      #"AV-31.36"(LOCK := #lock, ERR_EXTERN :=, LIOP_SEL := #Init, L_AUT := #Init, L_REMOTE := #Init, L_SIM :=, L_RESET := #Reset, AUT_OP :=, MAN_OP :=, SIM_OP :=, FB_OPEN :=, FB_CLOSE :=, L_MON := #Init, MON_T :=, MON_T_CLOSE :=, INSTANCE := 'AV-31.36', RESTART :=, VISIBILITY :=, OPdwCmd :=, QdwState =>, QwState =>, QCLOSING =>, QCLOSE =>, QOPENING =>, QOPEN =>, QCMD_OP =>, QMON =>, QMON_ERR =>, QMON_T =>, QMON_T_CLOSE =>, QMAN_AUT =>, QREMOTE =>, QSIM =>, QLOCK =>, QERR =>, QERR_EXT =>, QwAlarm =>)
   END_RUNG
   // the same network as SCL:
   #"AV-31.36"(LOCK := #lock,   // "Valve"
               LIOP_SEL := #Init,
               L_AUT := #Init,
               L_REMOTE := #Init,
               L_RESET := #Reset,
               L_MON := #Init,
               INSTANCE := 'AV-31.36');
END_REGION

REGION Network 117: AV-31.37
   RUNG wire#powerrail
      #"AV-31.37"(LOCK := #lock, ERR_EXTERN :=, LIOP_SEL := #Init, L_AUT := #Init, L_REMOTE := #Init, L_SIM :=, L_RESET := #Reset, AUT_OP :=, MAN_OP :=, SIM_OP :=, FB_OPEN :=, FB_CLOSE :=, L_MON := #Init, MON_T :=, MON_T_CLOSE :=, INSTANCE := 'AV-31.37', RESTART :=, VISIBILITY :=, OPdwCmd :=, QdwState =>, QwState =>, QCLOSING =>, QCLOSE =>, QOPENING =>, QOPEN =>, QCMD_OP =>, QMON =>, QMON_ERR =>, QMON_T =>, QMON_T_CLOSE =>, QMAN_AUT =>, QREMOTE =>, QSIM =>, QLOCK =>, QERR =>, QERR_EXT =>, QwAlarm =>)
   END_RUNG
   // the same network as SCL:
   #"AV-31.37"(LOCK := #lock,   // "Valve"
               LIOP_SEL := #Init,
               L_AUT := #Init,
               L_REMOTE := #Init,
               L_RESET := #Reset,
               L_MON := #Init,
               INSTANCE := 'AV-31.37');
END_REGION

REGION Network 118: AV-31.38
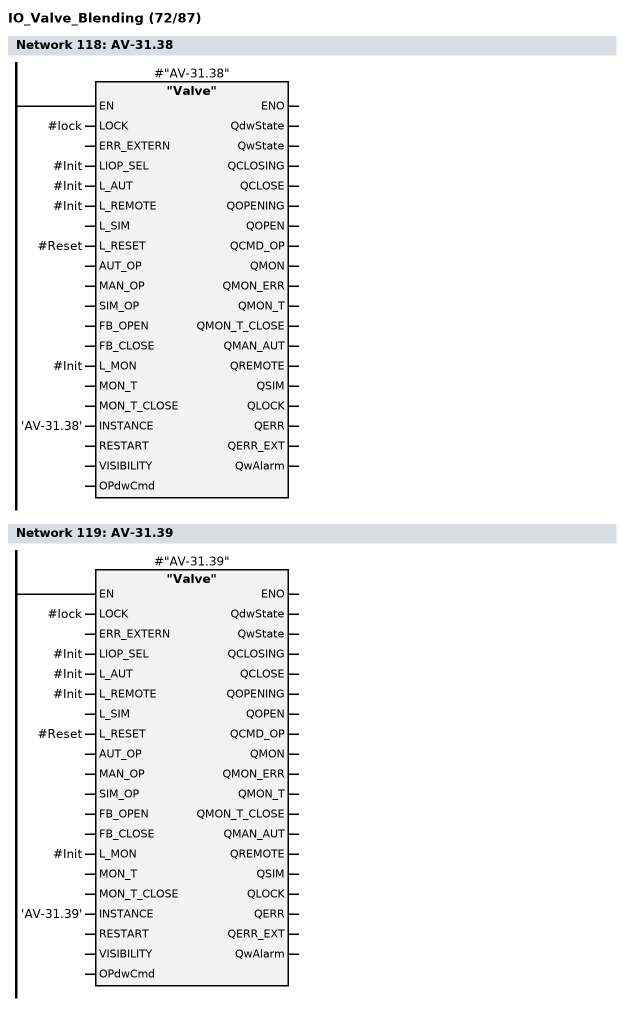
   RUNG wire#powerrail
      #"AV-31.38"(LOCK := #lock, ERR_EXTERN :=, LIOP_SEL := #Init, L_AUT := #Init, L_REMOTE := #Init, L_SIM :=, L_RESET := #Reset, AUT_OP :=, MAN_OP :=, SIM_OP :=, FB_OPEN :=, FB_CLOSE :=, L_MON := #Init, MON_T :=, MON_T_CLOSE :=, INSTANCE := 'AV-31.38', RESTART :=, VISIBILITY :=, OPdwCmd :=, QdwState =>, QwState =>, QCLOSING =>, QCLOSE =>, QOPENING =>, QOPEN =>, QCMD_OP =>, QMON =>, QMON_ERR =>, QMON_T =>, QMON_T_CLOSE =>, QMAN_AUT =>, QREMOTE =>, QSIM =>, QLOCK =>, QERR =>, QERR_EXT =>, QwAlarm =>)
   END_RUNG
   // the same network as SCL:
   #"AV-31.38"(LOCK := #lock,   // "Valve"
               LIOP_SEL := #Init,
               L_AUT := #Init,
               L_REMOTE := #Init,
               L_RESET := #Reset,
               L_MON := #Init,
               INSTANCE := 'AV-31.38');
END_REGION

REGION Network 119: AV-31.39
   RUNG wire#powerrail
      #"AV-31.39"(LOCK := #lock, ERR_EXTERN :=, LIOP_SEL := #Init, L_AUT := #Init, L_REMOTE := #Init, L_SIM :=, L_RESET := #Reset, AUT_OP :=, MAN_OP :=, SIM_OP :=, FB_OPEN :=, FB_CLOSE :=, L_MON := #Init, MON_T :=, MON_T_CLOSE :=, INSTANCE := 'AV-31.39', RESTART :=, VISIBILITY :=, OPdwCmd :=, QdwState =>, QwState =>, QCLOSING =>, QCLOSE =>, QOPENING =>, QOPEN =>, QCMD_OP =>, QMON =>, QMON_ERR =>, QMON_T =>, QMON_T_CLOSE =>, QMAN_AUT =>, QREMOTE =>, QSIM =>, QLOCK =>, QERR =>, QERR_EXT =>, QwAlarm =>)
   END_RUNG
   // the same network as SCL:
   #"AV-31.39"(LOCK := #lock,   // "Valve"
               LIOP_SEL := #Init,
               L_AUT := #Init,
               L_REMOTE := #Init,
               L_RESET := #Reset,
               L_MON := #Init,
               INSTANCE := 'AV-31.39');
END_REGION

REGION Network 120: AV-31.40
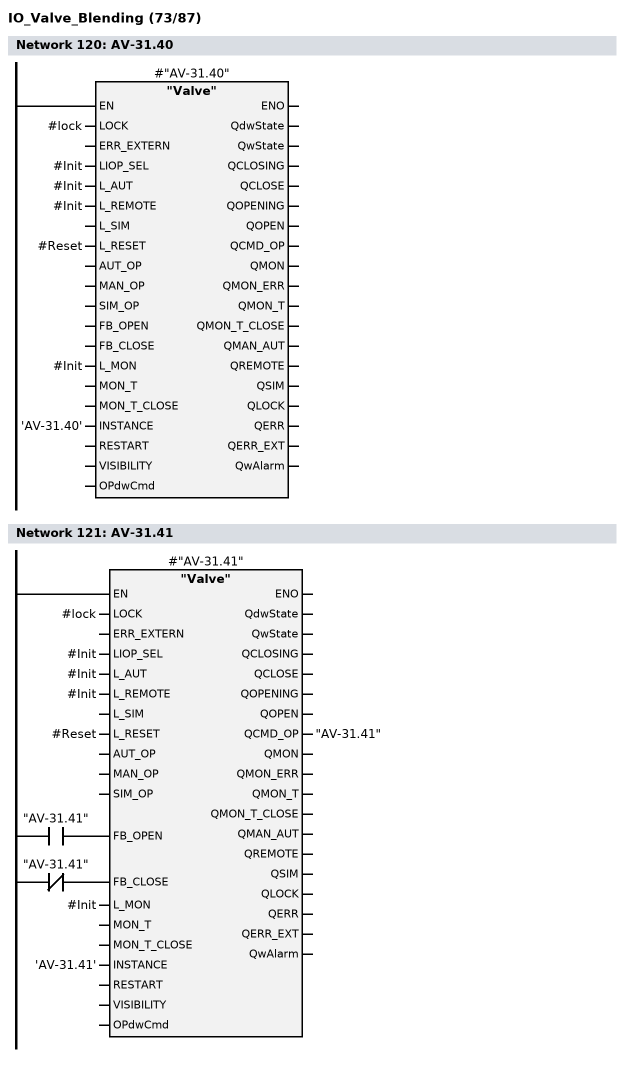
   RUNG wire#powerrail
      #"AV-31.40"(LOCK := #lock, ERR_EXTERN :=, LIOP_SEL := #Init, L_AUT := #Init, L_REMOTE := #Init, L_SIM :=, L_RESET := #Reset, AUT_OP :=, MAN_OP :=, SIM_OP :=, FB_OPEN :=, FB_CLOSE :=, L_MON := #Init, MON_T :=, MON_T_CLOSE :=, INSTANCE := 'AV-31.40', RESTART :=, VISIBILITY :=, OPdwCmd :=, QdwState =>, QwState =>, QCLOSING =>, QCLOSE =>, QOPENING =>, QOPEN =>, QCMD_OP =>, QMON =>, QMON_ERR =>, QMON_T =>, QMON_T_CLOSE =>, QMAN_AUT =>, QREMOTE =>, QSIM =>, QLOCK =>, QERR =>, QERR_EXT =>, QwAlarm =>)
   END_RUNG
   // the same network as SCL:
   #"AV-31.40"(LOCK := #lock,   // "Valve"
               LIOP_SEL := #Init,
               L_AUT := #Init,
               L_REMOTE := #Init,
               L_RESET := #Reset,
               L_MON := #Init,
               INSTANCE := 'AV-31.40');
END_REGION

REGION Network 121: AV-31.41
   RUNG wire#powerrail
      #"AV-31.41"(FB_OPEN := wire#w1, FB_CLOSE := wire#w2, LOCK := #lock, ERR_EXTERN :=, LIOP_SEL := #Init, L_AUT := #Init, L_REMOTE := #Init, L_SIM :=, L_RESET := #Reset, AUT_OP :=, MAN_OP :=, SIM_OP :=, L_MON := #Init, MON_T :=, MON_T_CLOSE :=, INSTANCE := 'AV-31.41', RESTART :=, VISIBILITY :=, OPdwCmd :=, QdwState =>, QwState =>, QCLOSING =>, QCLOSE =>, QOPENING =>, QOPEN =>, QCMD_OP => "AV-31.41", QMON =>, QMON_ERR =>, QMON_T =>, QMON_T_CLOSE =>, QMAN_AUT =>, QREMOTE =>, QSIM =>, QLOCK =>, QERR =>, QERR_EXT =>, QwAlarm =>)
   END_RUNG
   RUNG wire#powerrail
      Contact( "AV-31.41" )
   END_RUNG wire#w1
   RUNG wire#powerrail
      I_Contact( "AV-31.41" )
   END_RUNG wire#w2
   // the same network as SCL:
   #"AV-31.41"(LOCK := #lock,   // "Valve"
               LIOP_SEL := #Init,
               L_AUT := #Init,
               L_REMOTE := #Init,
               L_RESET := #Reset,
               FB_OPEN := "AV-31.41",
               FB_CLOSE := NOT "AV-31.41",
               L_MON := #Init,
               INSTANCE := 'AV-31.41',
               QCMD_OP => "AV-31.41");
END_REGION

REGION Network 122: AV-31.51
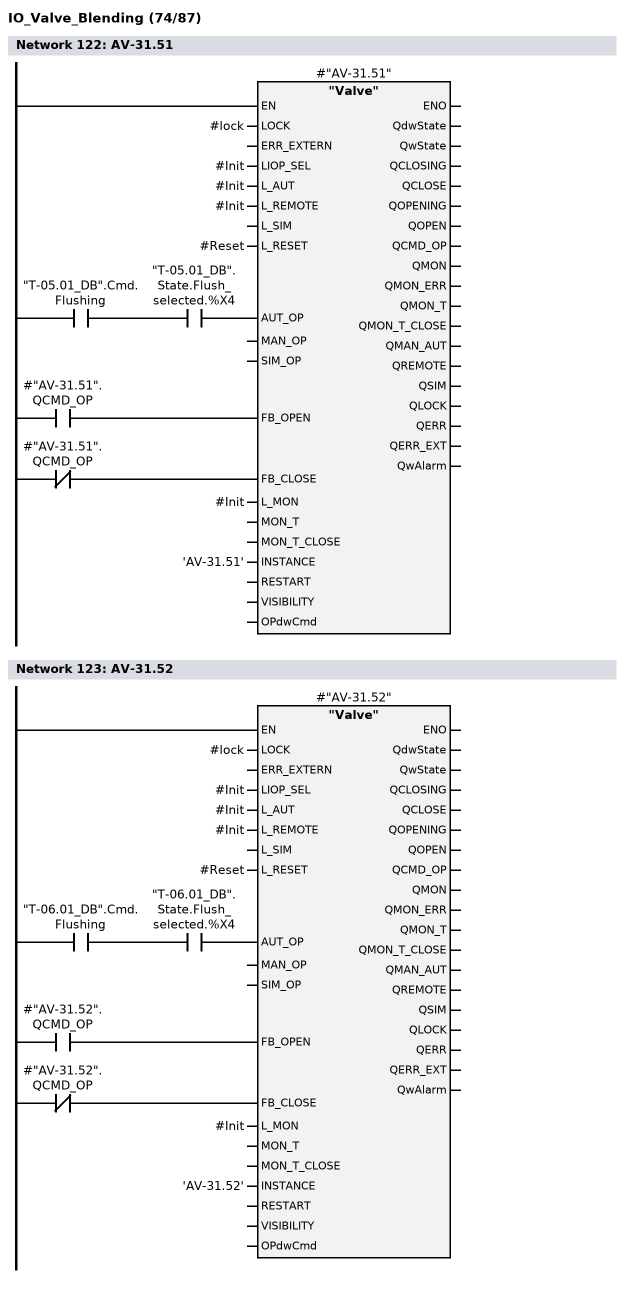
   RUNG wire#powerrail
      #"AV-31.51"(AUT_OP := wire#w1, FB_OPEN := wire#w2, FB_CLOSE := wire#w3, LOCK := #lock, ERR_EXTERN :=, LIOP_SEL := #Init, L_AUT := #Init, L_REMOTE := #Init, L_SIM :=, L_RESET := #Reset, MAN_OP :=, SIM_OP :=, L_MON := #Init, MON_T :=, MON_T_CLOSE :=, INSTANCE := 'AV-31.51', RESTART :=, VISIBILITY :=, OPdwCmd :=, QdwState =>, QwState =>, QCLOSING =>, QCLOSE =>, QOPENING =>, QOPEN =>, QCMD_OP =>, QMON =>, QMON_ERR =>, QMON_T =>, QMON_T_CLOSE =>, QMAN_AUT =>, QREMOTE =>, QSIM =>, QLOCK =>, QERR =>, QERR_EXT =>, QwAlarm =>)
   END_RUNG
   RUNG wire#powerrail
      Contact( "T-05.01_DB".Cmd.Flushing )
      Contact( "T-05.01_DB".State.Flush_selected.%X4 )
   END_RUNG wire#w1
   RUNG wire#powerrail
      Contact( #"AV-31.51".QCMD_OP )
   END_RUNG wire#w2
   RUNG wire#powerrail
      I_Contact( #"AV-31.51".QCMD_OP )
   END_RUNG wire#w3
   // the same network as SCL:
   #"AV-31.51"(LOCK := #lock,   // "Valve"
               LIOP_SEL := #Init,
               L_AUT := #Init,
               L_REMOTE := #Init,
               L_RESET := #Reset,
               AUT_OP := "T-05.01_DB".Cmd.Flushing AND "T-05.01_DB".State.Flush_selected.%X4,
               FB_OPEN := #"AV-31.51".QCMD_OP,
               FB_CLOSE := NOT #"AV-31.51".QCMD_OP,
               L_MON := #Init,
               INSTANCE := 'AV-31.51');
END_REGION

REGION Network 123: AV-31.52
   RUNG wire#powerrail
      #"AV-31.52"(AUT_OP := wire#w1, FB_OPEN := wire#w2, FB_CLOSE := wire#w3, LOCK := #lock, ERR_EXTERN :=, LIOP_SEL := #Init, L_AUT := #Init, L_REMOTE := #Init, L_SIM :=, L_RESET := #Reset, MAN_OP :=, SIM_OP :=, L_MON := #Init, MON_T :=, MON_T_CLOSE :=, INSTANCE := 'AV-31.52', RESTART :=, VISIBILITY :=, OPdwCmd :=, QdwState =>, QwState =>, QCLOSING =>, QCLOSE =>, QOPENING =>, QOPEN =>, QCMD_OP =>, QMON =>, QMON_ERR =>, QMON_T =>, QMON_T_CLOSE =>, QMAN_AUT =>, QREMOTE =>, QSIM =>, QLOCK =>, QERR =>, QERR_EXT =>, QwAlarm =>)
   END_RUNG
   RUNG wire#powerrail
      Contact( "T-06.01_DB".Cmd.Flushing )
      Contact( "T-06.01_DB".State.Flush_selected.%X4 )
   END_RUNG wire#w1
   RUNG wire#powerrail
      Contact( #"AV-31.52".QCMD_OP )
   END_RUNG wire#w2
   RUNG wire#powerrail
      I_Contact( #"AV-31.52".QCMD_OP )
   END_RUNG wire#w3
   // the same network as SCL:
   #"AV-31.52"(LOCK := #lock,   // "Valve"
               LIOP_SEL := #Init,
               L_AUT := #Init,
               L_REMOTE := #Init,
               L_RESET := #Reset,
               AUT_OP := "T-06.01_DB".Cmd.Flushing AND "T-06.01_DB".State.Flush_selected.%X4,
               FB_OPEN := #"AV-31.52".QCMD_OP,
               FB_CLOSE := NOT #"AV-31.52".QCMD_OP,
               L_MON := #Init,
               INSTANCE := 'AV-31.52');
END_REGION

REGION Network 124: AV-31.53
